LIN {X 0,Y 175.493,Z 504.64,A -85,B 0,C 180,E1 -23519.914,E2 -23519.914} C_VEL
LIN {X 0,Y 175.421,Z 500.697,A -85,B 0,C 180,E1 -23521.362,E2 -23521.362} C_VEL
LIN {X 0,Y 174.535,Z 496.874,A -85,B 0,C 180,E1 -23522.837,E2 -23522.837} C_VEL
LIN {X 0,Y 173.048,Z 491.549,A -85,B 0,C 180,E1 -23524.809,E2 -23524.809} C_VEL
LIN {X 0,Y 172.478,Z 487.181,A -85,B 0,C 180,E1 -23526.194,E2 -23526.194} C_VEL
LIN {X 0,Y 172.504,Z 485.618,A -85,B 0,C 180,E1 -23526.619,E2 -23526.619} C_VEL
LIN {X 0,Y 172.737,Z 474.589,A -85,B 0,C 180,E1 -23529.373,E2 -23529.373} C_VEL
LIN {X 0,Y 172.189,Z 465.013,A -85,B 0,C 180,E1 -23531.567,E2 -23531.567} C_VEL
LIN {X 0,Y 171.174,Z 457.609,A -85,B 0,C 180,E1 -23533.216,E2 -23533.216} C_VEL
LIN {X 0,Y 168.739,Z 450.808,A -85,B 0,C 180,E1 -23535.077,E2 -23535.077} C_VEL
LIN {X 0,Y 164.618,Z 441.913,A -85,B 0,C 180,E1 -23537.724,E2 -23537.724} C_VEL
LIN {X 0,Y 162.473,Z 437.771,A -85,B 0,C 180,E1 -23539.043,E2 -23539.043} C_VEL
LIN {X 0,Y 161.542,Z 436.333,A -85,B 0,C 180,E1 -23539.565,E2 -23539.565} C_VEL
LIN {X 0,Y 159.595,Z 433.029,A -85,B 0,C 180,E1 -23540.726,E2 -23540.726} C_VEL
LIN {X 0,Y 159.065,Z 431.216,A -85,B 0,C 180,E1 -23541.182,E2 -23541.182} C_VEL
LIN {X 0,Y 158.472,Z 427.771,A -85,B 0,C 180,E1 -23547.418,E2 -23547.418} C_VEL
LIN {X 0,Y 158.056,Z 424.721,A -85,B 0,C 180,E1 -23553.599,E2 -23553.599} C_VEL
LIN {X 0,Y 157.656,Z 422.287,A -85,B 0,C 180,E1 -23559.413,E2 -23559.413} C_VEL
LIN {X 0,Y 157.505,Z 421.4,A -85,B 0,C 180,E1 -23561.799,E2 -23561.799} C_VEL
LIN {X 0,Y 157.48,Z 420.87,A -85,B 0,C 180,E1 -23564.469,E2 -23564.469} C_VEL
LIN {X 0,Y 157.774,Z 420.833,A -85,B 0,C 180,E1 -23569.736,E2 -23569.736} C_VEL
LIN {X 0,Y 157.827,Z 420.827,A -85,B 0,C 180,E1 -23572.323,E2 -23572.323} C_VEL
LIN {X 0,Y 158.262,Z 420.771,A -85,B 0,C 180,E1 -23580,E2 -23580} C_VEL
LIN {X 0,Y 157.827,Z 420.823,A -85,B 0,C 180,E1 -23587.677,E2 -23587.677} C_VEL
LIN {X 0,Y 157.707,Z 420.841,A -85,B 0,C 180,E1 -23591.363,E2 -23591.363} C_VEL
LIN {X 0,Y 157.48,Z 420.866,A -85,B 0,C 180,E1 -23595.532,E2 -23595.532} C_VEL
LIN {X 0,Y 157.369,Z 420.882,A -85,B 0,C 180,E1 -23600.933,E2 -23600.933} C_VEL
LIN {X 0,Y 157.31,Z 420.887,A -85,B 0,C 180,E1 -23606.681,E2 -23606.681} C_VEL
LIN {X 0,Y 157.277,Z 420.885,A -85,B 0,C 180,E1 -23612.427,E2 -23612.427} C_VEL
LIN {X 0,Y 157.252,Z 420.892,A -85,B 0,C 180,E1 -23617.475,E2 -23617.475} C_VEL
LIN {X 0,Y 157.23,Z 421.026,A -85,B 0,C 180,E1 -23618.265,E2 -23618.265} C_VEL
LIN {X 0,Y 158.236,Z 423.75,A -85,B 0,C 180,E1 -23619.044,E2 -23619.044} C_VEL
LIN {X 0,Y 160.601,Z 426.337,A -85,B 0,C 180,E1 -23620.395,E2 -23620.395} C_VEL
LIN {X 0,Y 162.443,Z 429.537,A -85,B 0,C 180,E1 -23621.594,E2 -23621.594} C_VEL
LIN {X 0,Y 163.808,Z 431.474,A -85,B 0,C 180,E1 -23622.408,E2 -23622.408} C_VEL
LIN {X 0,Y 168.225,Z 439.084,A -85,B 0,C 180,E1 -23625.253,E2 -23625.253} C_VEL
LIN {X 0,Y 171.385,Z 446.088,A -85,B 0,C 180,E1 -23627.572,E2 -23627.572} C_VEL
LIN {X 0,Y 174.009,Z 454.383,A -85,B 0,C 180,E1 -23630.12,E2 -23630.12} C_VEL
LIN {X 0,Y 175.758,Z 463.088,A -85,B 0,C 180,E1 -23632.727,E2 -23632.727} C_VEL
LIN {X 0,Y 176.597,Z 472.445,A -85,B 0,C 180,E1 -23635.6,E2 -23635.6} C_VEL
LIN {X 0,Y 176.668,Z 474.207,A -85,B 0,C 180,E1 -23636.156,E2 -23636.156} C_VEL
LIN {X 0,Y 174.39,Z 481.217,A -85,B 0,C 180,E1 -23638.023,E2 -23638.023} C_VEL
LIN {X 0,Y 170.562,Z 490.741,A -85,B 0,C 180,E1 -23641.043,E2 -23641.043} C_VEL
LIN {X 0,Y 166.711,Z 498.951,A -85,B 0,C 180,E1 -23644.399,E2 -23644.399} C_VEL
LIN {X 0,Y 164.054,Z 504.551,A -85,B 0,C 180,E1 -23647.322,E2 -23647.322} C_VEL
LIN {X 0,Y 161.243,Z 510.012,A -85,B 0,C 180,E1 -23650.92,E2 -23650.92} C_VEL
LIN {X 0,Y 158.999,Z 514.292,A -85,B 0,C 180,E1 -23654.621,E2 -23654.621} C_VEL
LIN {X 0,Y 157.864,Z 516.551,A -85,B 0,C 180,E1 -23657.139,E2 -23657.139} C_VEL
LIN {X 0,Y 156.746,Z 518.873,A -85,B 0,C 180,E1 -23660.546,E2 -23660.546} C_VEL
LIN {X 0,Y 155.819,Z 520.739,A -85,B 0,C 180,E1 -23664.825,E2 -23664.825} C_VEL
LIN {X 0,Y 155.405,Z 521.567,A -85,B 0,C 180,E1 -23670,E2 -23670} C_VEL
LIN {X 0,Y 155.514,Z 521.37,A -85,B 0,C 180,E1 -23672.59,E2 -23672.59} C_VEL
LIN {X 0,Y 155.811,Z 520.787,A -85,B 0,C 180,E1 -23675.176,E2 -23675.176} C_VEL
LIN {X 0,Y 156.94,Z 518.483,A -85,B 0,C 180,E1 -23680.319,E2 -23680.319} C_VEL
LIN {X 0,Y 158.342,Z 515.638,A -85,B 0,C 180,E1 -23684.13,E2 -23684.13} C_VEL
LIN {X 0,Y 160.383,Z 511.769,A -85,B 0,C 180,E1 -23687.863,E2 -23687.863} C_VEL
LIN {X 0,Y 162.981,Z 506.773,A -85,B 0,C 180,E1 -23691.502,E2 -23691.502} C_VEL
LIN {X 0,Y 166.065,Z 500.477,A -85,B 0,C 180,E1 -23695.038,E2 -23695.038} C_VEL
LIN {X 0,Y 169.842,Z 492.583,A -85,B 0,C 180,E1 -23698.416,E2 -23698.416} C_VEL
LIN {X 0,Y 173.954,Z 482.769,A -85,B 0,C 180,E1 -23701.684,E2 -23701.684} C_VEL
LIN {X 0,Y 176.747,Z 474.731,A -85,B 0,C 180,E1 -23703.827,E2 -23703.827} C_VEL
LIN {X 0,Y 176.346,Z 467.155,A -85,B 0,C 180,E1 -23706.194,E2 -23706.194} C_VEL
LIN {X 0,Y 174.874,Z 457.677,A -85,B 0,C 180,E1 -23709.05,E2 -23709.05} C_VEL
LIN {X 0,Y 172.59,Z 449.442,A -85,B 0,C 180,E1 -23711.56,E2 -23711.56} C_VEL
LIN {X 0,Y 170.161,Z 443.217,A -85,B 0,C 180,E1 -23713.554,E2 -23713.554} C_VEL
LIN {X 0,Y 165.724,Z 434.544,A -85,B 0,C 180,E1 -23716.601,E2 -23716.601} C_VEL
LIN {X 0,Y 163.507,Z 430.878,A -85,B 0,C 180,E1 -23718.016,E2 -23718.016} C_VEL
LIN {X 0,Y 160.947,Z 427.183,A -85,B 0,C 180,E1 -23719.565,E2 -23719.565} C_VEL
LIN {X 0,Y 160.394,Z 425.942,A -85,B 0,C 180,E1 -23719.971,E2 -23719.971} C_VEL
LIN {X 0,Y 158.165,Z 423.621,A -85,B 0,C 180,E1 -23721.234,E2 -23721.234} C_VEL
LIN {X 0,Y 157.222,Z 420.897,A -85,B 0,C 180,E1 -23722.046,E2 -23722.046} C_VEL
LIN {X 0,Y 157.292,Z 420.884,A -85,B 0,C 180,E1 -23724.489,E2 -23724.489} C_VEL
LIN {X 0,Y 157.296,Z 420.89,A -85,B 0,C 180,E1 -23728.096,E2 -23728.096} C_VEL
LIN {X 0,Y 157.317,Z 420.889,A -85,B 0,C 180,E1 -23733.465,E2 -23733.465} C_VEL
LIN {X 0,Y 157.395,Z 420.879,A -85,B 0,C 180,E1 -23739.669,E2 -23739.669} C_VEL
LIN {X 0,Y 157.476,Z 420.869,A -85,B 0,C 180,E1 -23744.468,E2 -23744.468} C_VEL
LIN {X 0,Y 157.692,Z 420.84,A -85,B 0,C 180,E1 -23749.731,E2 -23749.731} C_VEL
LIN {X 0,Y 157.77,Z 420.831,A -85,B 0,C 180,E1 -23752.32,E2 -23752.32} C_VEL
LIN {X 0,Y 158.261,Z 420.776,A -85,B 0,C 180,E1 -23760,E2 -23760} C_VEL
LIN {X 0,Y 157.828,Z 420.829,A -85,B 0,C 180,E1 -23767.677,E2 -23767.677} C_VEL
LIN {X 0,Y 157.72,Z 420.838,A -85,B 0,C 180,E1 -23771.383,E2 -23771.383} C_VEL
LIN {X 0,Y 157.489,Z 420.866,A -85,B 0,C 180,E1 -23775.531,E2 -23775.531} C_VEL
LIN {X 0,Y 157.542,Z 421.446,A -85,B 0,C 180,E1 -23778.196,E2 -23778.196} C_VEL
LIN {X 0,Y 157.82,Z 423.583,A -85,B 0,C 180,E1 -23783.627,E2 -23783.627} C_VEL
LIN {X 0,Y 158.101,Z 425.177,A -85,B 0,C 180,E1 -23787.244,E2 -23787.244} C_VEL
LIN {X 0,Y 158.474,Z 427.834,A -85,B 0,C 180,E1 -23792.582,E2 -23792.582} C_VEL
LIN {X 0,Y 159.063,Z 431.245,A -85,B 0,C 180,E1 -23798.717,E2 -23798.717} C_VEL
LIN {X 0,Y 160.489,Z 434.863,A -85,B 0,C 180,E1 -23799.723,E2 -23799.723} C_VEL
LIN {X 0,Y 162.468,Z 437.655,A -85,B 0,C 180,E1 -23800.825,E2 -23800.825} C_VEL
LIN {X 0,Y 164.462,Z 441.653,A -85,B 0,C 180,E1 -23802.073,E2 -23802.073} C_VEL
LIN {X 0,Y 165.475,Z 443.522,A -85,B 0,C 180,E1 -23802.676,E2 -23802.676} C_VEL
LIN {X 0,Y 168.043,Z 449.265,A -85,B 0,C 180,E1 -23804.365,E2 -23804.365} C_VEL
LIN {X 0,Y 170.827,Z 456.275,A -85,B 0,C 180,E1 -23806.35,E2 -23806.35} C_VEL
LIN {X 0,Y 172.062,Z 463.231,A -85,B 0,C 180,E1 -23807.965,E2 -23807.965} C_VEL
LIN {X 0,Y 172.805,Z 473.587,A -85,B 0,C 180,E1 -23810.33,E2 -23810.33} C_VEL
LIN {X 0,Y 172.705,Z 483.558,A -85,B 0,C 180,E1 -23812.784,E2 -23812.784} C_VEL
LIN {X 0,Y 171.722,Z 494.309,A -85,B 0,C 180,E1 -23815.754,E2 -23815.754} C_VEL
LIN {X 0,Y 170.269,Z 502.262,A -85,B 0,C 180,E1 -23818.246,E2 -23818.246} C_VEL
LIN {X 0,Y 168.438,Z 507.397,A -85,B 0,C 180,E1 -23819.953,E2 -23819.953} C_VEL
LIN {X 0,Y 165.157,Z 514.724,A -85,B 0,C 180,E1 -23822.777,E2 -23822.777} C_VEL
LIN {X 0,Y 162.483,Z 520.901,A -85,B 0,C 180,E1 -23825.773,E2 -23825.773} C_VEL
LIN {X 0,Y 159.679,Z 526.854,A -85,B 0,C 180,E1 -23829.383,E2 -23829.383} C_VEL
LIN {X 0,Y 157.532,Z 531.619,A -85,B 0,C 180,E1 -23833.142,E2 -23833.142} C_VEL
LIN {X 0,Y 156.082,Z 535.276,A -85,B 0,C 180,E1 -23836.989,E2 -23836.989} C_VEL
LIN {X 0,Y 155.465,Z 537.169,A -85,B 0,C 180,E1 -23839.582,E2 -23839.582} C_VEL
LIN {X 0,Y 155.141,Z 538.598,A -85,B 0,C 180,E1 -23842.189,E2 -23842.189} C_VEL
LIN {X 0,Y 155.009,Z 539.965,A -85,B 0,C 180,E1 -23845.92,E2 -23845.92} C_VEL
LIN {X 0,Y 155.237,Z 540.486,A -85,B 0,C 180,E1 -23850,E2 -23850} C_VEL
LIN {X 0,Y 155.013,Z 539.948,A -85,B 0,C 180,E1 -23854.1,E2 -23854.1} C_VEL
LIN {X 0,Y 155.113,Z 538.571,A -85,B 0,C 180,E1 -23857.812,E2 -23857.812} C_VEL
LIN {X 0,Y 155.463,Z 537.132,A -85,B 0,C 180,E1 -23860.418,E2 -23860.418} C_VEL
LIN {X 0,Y 156.466,Z 534.131,A -85,B 0,C 180,E1 -23864.302,E2 -23864.302} C_VEL
LIN {X 0,Y 158.189,Z 530.096,A -85,B 0,C 180,E1 -23868.119,E2 -23868.119} C_VEL
LIN {X 0,Y 161.039,Z 523.913,A -85,B 0,C 180,E1 -23872.449,E2 -23872.449} C_VEL
LIN {X 0,Y 164.023,Z 517.168,A -85,B 0,C 180,E1 -23876.052,E2 -23876.052} C_VEL
LIN {X 0,Y 167.699,Z 508.823,A -85,B 0,C 180,E1 -23879.5,E2 -23879.5} C_VEL
LIN {X 0,Y 169.803,Z 503.886,A -85,B 0,C 180,E1 -23881.156,E2 -23881.156} C_VEL
LIN {X 0,Y 171.491,Z 495.166,A -85,B 0,C 180,E1 -23883.944,E2 -23883.944} C_VEL
LIN {X 0,Y 172.504,Z 485.618,A -85,B 0,C 180,E1 -23886.619,E2 -23886.619} C_VEL
LIN {X 0,Y 172.159,Z 481.183,A -85,B 0,C 180,E1 -23887.899,E2 -23887.899} C_VEL
LIN {X 0,Y 170.903,Z 477.034,A -85,B 0,C 180,E1 -23889.266,E2 -23889.266} C_VEL
LIN {X 0,Y 167.544,Z 468.986,A -85,B 0,C 180,E1 -23892.064,E2 -23892.064} C_VEL
LIN {X 0,Y 166.046,Z 462.962,A -85,B 0,C 180,E1 -23893.79,E2 -23893.79} C_VEL
LIN {X 0,Y 165.199,Z 458.874,A -85,B 0,C 180,E1 -23894.864,E2 -23894.864} C_VEL
LIN {X 0,Y 162.424,Z 451.6,A -85,B 0,C 180,E1 -23897.123,E2 -23897.123} C_VEL
LIN {X 0,Y 159.982,Z 446.385,A -85,B 0,C 180,E1 -23898.885,E2 -23898.885} C_VEL
LIN {X 0,Y 157.628,Z 441.579,A -85,B 0,C 180,E1 -23900.554,E2 -23900.554} C_VEL
LIN {X 0,Y 155.555,Z 437.698,A -85,B 0,C 180,E1 -23902.001,E2 -23902.001} C_VEL
LIN {X 0,Y 154.89,Z 436.44,A -85,B 0,C 180,E1 -23902.456,E2 -23902.456} C_VEL
LIN {X 0,Y 152.505,Z 433.06,A -85,B 0,C 180,E1 -23904.015,E2 -23904.015} C_VEL
LIN {X 0,Y 151.729,Z 430.582,A -85,B 0,C 180,E1 -23904.722,E2 -23904.722} C_VEL
LIN {X 0,Y 151.32,Z 428.28,A -85,B 0,C 180,E1 -23909.277,E2 -23909.277} C_VEL
LIN {X 0,Y 151.168,Z 426.831,A -85,B 0,C 180,E1 -23912.295,E2 -23912.295} C_VEL
LIN {X 0,Y 150.769,Z 424.399,A -85,B 0,C 180,E1 -23918.105,E2 -23918.105} C_VEL
LIN {X 0,Y 150.494,Z 422.416,A -85,B 0,C 180,E1 -23923.728,E2 -23923.728} C_VEL
LIN {X 0,Y 150.466,Z 421.744,A -85,B 0,C 180,E1 -23926.494,E2 -23926.494} C_VEL
LIN {X 0,Y 150.697,Z 421.715,A -85,B 0,C 180,E1 -23929.249,E2 -23929.249} C_VEL
LIN {X 0,Y 150.765,Z 421.706,A -85,B 0,C 180,E1 -23931.961,E2 -23931.961} C_VEL
LIN {X 0,Y 151.222,Z 421.648,A -85,B 0,C 180,E1 -23940,E2 -23940} C_VEL
LIN {X 0,Y 150.765,Z 421.704,A -85,B 0,C 180,E1 -23948.039,E2 -23948.039} C_VEL
LIN {X 0,Y 150.637,Z 421.722,A -85,B 0,C 180,E1 -23951.546,E2 -23951.546} C_VEL
LIN {X 0,Y 150.385,Z 421.75,A -85,B 0,C 180,E1 -23956.284,E2 -23956.284} C_VEL
LIN {X 0,Y 150.351,Z 421.756,A -85,B 0,C 180,E1 -23960.791,E2 -23960.791} C_VEL
LIN {X 0,Y 150.242,Z 421.768,A -85,B 0,C 180,E1 -23967.28,E2 -23967.28} C_VEL
LIN {X 0,Y 150.217,Z 421.764,A -85,B 0,C 180,E1 -23972.633,E2 -23972.633} C_VEL
LIN {X 0,Y 150.234,Z 421.892,A -85,B 0,C 180,E1 -23974.76,E2 -23974.76} C_VEL
LIN {X 0,Y 151.187,Z 424.529,A -85,B 0,C 180,E1 -23975.628,E2 -23975.628} C_VEL
LIN {X 0,Y 153.348,Z 426.792,A -85,B 0,C 180,E1 -23977.056,E2 -23977.056} C_VEL
LIN {X 0,Y 155.822,Z 430.828,A -85,B 0,C 180,E1 -23978.864,E2 -23978.864} C_VEL
LIN {X 0,Y 156.885,Z 432.163,A -85,B 0,C 180,E1 -23979.566,E2 -23979.566} C_VEL
LIN {X 0,Y 160.888,Z 438.893,A -85,B 0,C 180,E1 -23982.446,E2 -23982.446} C_VEL
LIN {X 0,Y 164.275,Z 445.344,A -85,B 0,C 180,E1 -23984.992,E2 -23984.992} C_VEL
LIN {X 0,Y 166.93,Z 452.435,A -85,B 0,C 180,E1 -23987.46,E2 -23987.46} C_VEL
LIN {X 0,Y 168.941,Z 460.421,A -85,B 0,C 180,E1 -23990.069,E2 -23990.069} C_VEL
LIN {X 0,Y 170.032,Z 468.449,A -85,B 0,C 180,E1 -23992.662,E2 -23992.662} C_VEL
LIN {X 0,Y 170.291,Z 476.562,A -85,B 0,C 180,E1 -23995.361,E2 -23995.361} C_VEL
LIN {X 0,Y 166.541,Z 486.299,A -85,B 0,C 180,E1 -23998.163,E2 -23998.163} C_VEL
LIN {X 0,Y 162.992,Z 494.122,A -85,B 0,C 180,E1 -24000.982,E2 -24000.982} C_VEL
LIN {X 0,Y 159.238,Z 501.757,A -85,B 0,C 180,E1 -24004.512,E2 -24004.512} C_VEL
LIN {X 0,Y 155.5,Z 508.765,A -85,B 0,C 180,E1 -24008.804,E2 -24008.804} C_VEL
LIN {X 0,Y 152.899,Z 513.427,A -85,B 0,C 180,E1 -24012.616,E2 -24012.616} C_VEL
LIN {X 0,Y 150.96,Z 516.984,A -85,B 0,C 180,E1 -24016.54,E2 -24016.54} C_VEL
LIN {X 0,Y 149.624,Z 519.54,A -85,B 0,C 180,E1 -24020.539,E2 -24020.539} C_VEL
LIN {X 0,Y 148.769,Z 521.17,A -85,B 0,C 180,E1 -24024.579,E2 -24024.579} C_VEL
LIN {X 0,Y 148.465,Z 521.771,A -85,B 0,C 180,E1 -24027.287,E2 -24027.287} C_VEL
LIN {X 0,Y 148.346,Z 521.997,A -85,B 0,C 180,E1 -24030,E2 -24030} C_VEL
LIN {X 0,Y 148.462,Z 521.8,A -85,B 0,C 180,E1 -24032.714,E2 -24032.714} C_VEL
LIN {X 0,Y 148.76,Z 521.218,A -85,B 0,C 180,E1 -24035.422,E2 -24035.422} C_VEL
LIN {X 0,Y 149.979,Z 518.913,A -85,B 0,C 180,E1 -24040.804,E2 -24040.804} C_VEL
LIN {X 0,Y 151.475,Z 516.069,A -85,B 0,C 180,E1 -24044.785,E2 -24044.785} C_VEL
LIN {X 0,Y 153.644,Z 512.2,A -85,B 0,C 180,E1 -24048.675,E2 -24048.675} C_VEL
LIN {X 0,Y 156.409,Z 507.203,A -85,B 0,C 180,E1 -24052.454,E2 -24052.454} C_VEL
LIN {X 0,Y 159.667,Z 500.906,A -85,B 0,C 180,E1 -24056.115,E2 -24056.115} C_VEL
LIN {X 0,Y 163.653,Z 493.011,A -85,B 0,C 180,E1 -24059.595,E2 -24059.595} C_VEL
LIN {X 0,Y 167.954,Z 483.198,A -85,B 0,C 180,E1 -24062.956,E2 -24062.956} C_VEL
LIN {X 0,Y 170.483,Z 476.31,A -85,B 0,C 180,E1 -24064.859,E2 -24064.859} C_VEL
LIN {X 0,Y 170.175,Z 468.722,A -85,B 0,C 180,E1 -24067.401,E2 -24067.401} C_VEL
LIN {X 0,Y 168.987,Z 460.08,A -85,B 0,C 180,E1 -24070.194,E2 -24070.194} C_VEL
LIN {X 0,Y 167.089,Z 452.794,A -85,B 0,C 180,E1 -24072.6,E2 -24072.6} C_VEL
LIN {X 0,Y 164.806,Z 446.556,A -85,B 0,C 180,E1 -24074.781,E2 -24074.781} C_VEL
LIN {X 0,Y 161.086,Z 439.296,A -85,B 0,C 180,E1 -24077.618,E2 -24077.618} C_VEL
LIN {X 0,Y 156.396,Z 431.427,A -85,B 0,C 180,E1 -24081.014,E2 -24081.014} C_VEL
LIN {X 0,Y 154.307,Z 428.597,A -85,B 0,C 180,E1 -24082.434,E2 -24082.434} C_VEL
LIN {X 0,Y 153.487,Z 426.898,A -85,B 0,C 180,E1 -24083.103,E2 -24083.103} C_VEL
LIN {X 0,Y 151.343,Z 424.737,A -85,B 0,C 180,E1 -24084.516,E2 -24084.516} C_VEL
LIN {X 0,Y 150.258,Z 422.177,A -85,B 0,C 180,E1 -24085.45,E2 -24085.45} C_VEL
LIN {X 0,Y 150.206,Z 421.769,A -85,B 0,C 180,E1 -24085.64,E2 -24085.64} C_VEL
LIN {X 0,Y 150.209,Z 421.775,A -85,B 0,C 180,E1 -24089.024,E2 -24089.024} C_VEL
LIN {X 0,Y 150.243,Z 421.768,A -85,B 0,C 180,E1 -24092.721,E2 -24092.721} C_VEL
LIN {X 0,Y 150.352,Z 421.757,A -85,B 0,C 180,E1 -24099.209,E2 -24099.209} C_VEL
LIN {X 0,Y 150.382,Z 421.75,A -85,B 0,C 180,E1 -24103.715,E2 -24103.715} C_VEL
LIN {X 0,Y 150.615,Z 421.721,A -85,B 0,C 180,E1 -24109.243,E2 -24109.243} C_VEL
LIN {X 0,Y 150.707,Z 421.711,A -85,B 0,C 180,E1 -24111.958,E2 -24111.958} C_VEL
LIN {X 0,Y 151.221,Z 421.654,A -85,B 0,C 180,E1 -24120,E2 -24120} C_VEL
LIN {X 0,Y 150.767,Z 421.709,A -85,B 0,C 180,E1 -24128.039,E2 -24128.039} C_VEL
LIN {X 0,Y 150.645,Z 421.719,A -85,B 0,C 180,E1 -24131.56,E2 -24131.56} C_VEL
LIN {X 0,Y 150.47,Z 421.741,A -85,B 0,C 180,E1 -24133.505,E2 -24133.505} C_VEL
LIN {X 0,Y 150.665,Z 423.414,A -85,B 0,C 180,E1 -24139.058,E2 -24139.058} C_VEL
LIN {X 0,Y 150.946,Z 425.635,A -85,B 0,C 180,E1 -24144.774,E2 -24144.774} C_VEL
LIN {X 0,Y 151.185,Z 427.018,A -85,B 0,C 180,E1 -24147.963,E2 -24147.963} C_VEL
LIN {X 0,Y 151.646,Z 430.268,A -85,B 0,C 180,E1 -24154.592,E2 -24154.592} C_VEL
LIN {X 0,Y 151.724,Z 430.738,A -85,B 0,C 180,E1 -24155.178,E2 -24155.178} C_VEL
LIN {X 0,Y 152.952,Z 433.942,A -85,B 0,C 180,E1 -24156.168,E2 -24156.168} C_VEL
LIN {X 0,Y 155.39,Z 437.231,A -85,B 0,C 180,E1 -24157.73,E2 -24157.73} C_VEL
LIN {X 0,Y 157.426,Z 441.33,A -85,B 0,C 180,E1 -24159.196,E2 -24159.196} C_VEL
LIN {X 0,Y 158.706,Z 443.64,A -85,B 0,C 180,E1 -24160.053,E2 -24160.053} C_VEL
LIN {X 0,Y 161.186,Z 448.748,A -85,B 0,C 180,E1 -24161.826,E2 -24161.826} C_VEL
LIN {X 0,Y 164.43,Z 456.664,A -85,B 0,C 180,E1 -24164.36,E2 -24164.36} C_VEL
LIN {X 0,Y 165.782,Z 460.967,A -85,B 0,C 180,E1 -24165.615,E2 -24165.615} C_VEL
LIN {X 0,Y 166.735,Z 470.398,A -85,B 0,C 180,E1 -24167.933,E2 -24167.933} C_VEL
LIN {X 0,Y 166.739,Z 481.622,A -85,B 0,C 180,E1 -24170.783,E2 -24170.783} C_VEL
LIN {X 0,Y 165.823,Z 491.754,A -85,B 0,C 180,E1 -24173.636,E2 -24173.636} C_VEL
LIN {X 0,Y 164.504,Z 499.99,A -85,B 0,C 180,E1 -24176.262,E2 -24176.262} C_VEL
LIN {X 0,Y 163.014,Z 505.323,A -85,B 0,C 180,E1 -24178.12,E2 -24178.12} C_VEL
LIN {X 0,Y 158.822,Z 514.29,A -85,B 0,C 180,E1 -24181.595,E2 -24181.595} C_VEL
LIN {X 0,Y 155.634,Z 521.247,A -85,B 0,C 180,E1 -24185.126,E2 -24185.126} C_VEL
LIN {X 0,Y 153.002,Z 526.42,A -85,B 0,C 180,E1 -24188.44,E2 -24188.44} C_VEL
LIN {X 0,Y 150.706,Z 531.185,A -85,B 0,C 180,E1 -24192.355,E2 -24192.355} C_VEL
LIN {X 0,Y 149.123,Z 534.841,A -85,B 0,C 180,E1 -24196.37,E2 -24196.37} C_VEL
LIN {X 0,Y 148.469,Z 536.736,A -85,B 0,C 180,E1 -24199.085,E2 -24199.085} C_VEL
LIN {X 0,Y 148.07,Z 538.164,A -85,B 0,C 180,E1 -24201.813,E2 -24201.813} C_VEL
LIN {X 0,Y 147.94,Z 539.595,A -85,B 0,C 180,E1 -24206.05,E2 -24206.05} C_VEL
LIN {X 0,Y 148.153,Z 540.054,A -85,B 0,C 180,E1 -24210,E2 -24210} C_VEL
LIN {X 0,Y 147.934,Z 539.59,A -85,B 0,C 180,E1 -24213.916,E2 -24213.916} C_VEL
LIN {X 0,Y 148.046,Z 538.136,A -85,B 0,C 180,E1 -24218.187,E2 -24218.187} C_VEL
LIN {X 0,Y 148.468,Z 536.698,A -85,B 0,C 180,E1 -24220.915,E2 -24220.915} C_VEL
LIN {X 0,Y 149.564,Z 533.695,A -85,B 0,C 180,E1 -24224.978,E2 -24224.978} C_VEL
LIN {X 0,Y 151.409,Z 529.659,A -85,B 0,C 180,E1 -24228.961,E2 -24228.961} C_VEL
LIN {X 0,Y 154.493,Z 523.478,A -85,B 0,C 180,E1 -24233.456,E2 -24233.456} C_VEL
LIN {X 0,Y 157.656,Z 516.732,A -85,B 0,C 180,E1 -24237.189,E2 -24237.189} C_VEL
LIN {X 0,Y 161.544,Z 508.387,A -85,B 0,C 180,E1 -24240.743,E2 -24240.743} C_VEL
LIN {X 0,Y 163.59,Z 503.438,A -85,B 0,C 180,E1 -24242.48,E2 -24242.48} C_VEL
LIN {X 0,Y 165.321,Z 494.743,A -85,B 0,C 180,E1 -24245.383,E2 -24245.383} C_VEL
LIN {X 0,Y 166.4,Z 485.318,A -85,B 0,C 180,E1 -24248.148,E2 -24248.148} C_VEL
LIN {X 0,Y 166.763,Z 474.342,A -85,B 0,C 180,E1 -24251.02,E2 -24251.02} C_VEL
LIN {X 0,Y 166.149,Z 463.815,A -85,B 0,C 180,E1 -24253.583,E2 -24253.583} C_VEL
LIN {X 0,Y 166.046,Z 462.962,A -85,B 0,C 180,E1 -24253.79,E2 -24253.79} C_VEL
LIN {X 0,Y 165.299,Z 460.01,A -85,B 0,C 180,E1 -24254.631,E2 -24254.631} C_VEL
LIN {X 0,Y 163.174,Z 456.37,A -85,B 0,C 180,E1 -24256.067,E2 -24256.067} C_VEL
LIN {X 0,Y 160.391,Z 453.439,A -85,B 0,C 180,E1 -24257.617,E2 -24257.617} C_VEL
LIN {X 0,Y 154.426,Z 447.845,A -85,B 0,C 180,E1 -24260.975,E2 -24260.975} C_VEL
LIN {X 0,Y 152.812,Z 445.559,A -85,B 0,C 180,E1 -24262.089,E2 -24262.089} C_VEL
LIN {X 0,Y 150.995,Z 441.721,A -85,B 0,C 180,E1 -24263.598,E2 -24263.598} C_VEL
LIN {X 0,Y 148.744,Z 437.9,A -85,B 0,C 180,E1 -24265.357,E2 -24265.357} C_VEL
LIN {X 0,Y 147.886,Z 436.021,A -85,B 0,C 180,E1 -24266.099,E2 -24266.099} C_VEL
LIN {X 0,Y 145.416,Z 432.796,A -85,B 0,C 180,E1 -24267.986,E2 -24267.986} C_VEL
LIN {X 0,Y 144.374,Z 429.792,A -85,B 0,C 180,E1 -24269.058,E2 -24269.058} C_VEL
LIN {X 0,Y 144.059,Z 427.599,A -85,B 0,C 180,E1 -24273.956,E2 -24273.956} C_VEL
LIN {X 0,Y 143.761,Z 425.302,A -85,B 0,C 180,E1 -24279.989,E2 -24279.989} C_VEL
LIN {X 0,Y 143.529,Z 423.451,A -85,B 0,C 180,E1 -24285.828,E2 -24285.828} C_VEL
LIN {X 0,Y 143.624,Z 422.621,A -85,B 0,C 180,E1 -24288.713,E2 -24288.713} C_VEL
LIN {X 0,Y 143.688,Z 422.587,A -85,B 0,C 180,E1 -24291.562,E2 -24291.562} C_VEL
LIN {X 0,Y 144.181,Z 422.525,A -85,B 0,C 180,E1 -24300,E2 -24300} C_VEL
LIN {X 0,Y 143.687,Z 422.588,A -85,B 0,C 180,E1 -24308.438,E2 -24308.438} C_VEL
LIN {X 0,Y 143.573,Z 422.602,A -85,B 0,C 180,E1 -24311.758,E2 -24311.758} C_VEL
LIN {X 0,Y 143.318,Z 422.633,A -85,B 0,C 180,E1 -24317.111,E2 -24317.111} C_VEL
LIN {X 0,Y 143.277,Z 422.636,A -85,B 0,C 180,E1 -24321.253,E2 -24321.253} C_VEL
LIN {X 0,Y 143.189,Z 422.649,A -85,B 0,C 180,E1 -24327.936,E2 -24327.936} C_VEL
LIN {X 0,Y 143.139,Z 422.68,A -85,B 0,C 180,E1 -24330.42,E2 -24330.42} C_VEL
LIN {X 0,Y 144.036,Z 425.274,A -85,B 0,C 180,E1 -24331.432,E2 -24331.432} C_VEL
LIN {X 0,Y 146.042,Z 427.52,A -85,B 0,C 180,E1 -24333.062,E2 -24333.062} C_VEL
LIN {X 0,Y 147.03,Z 428.412,A -85,B 0,C 180,E1 -24333.822,E2 -24333.822} C_VEL
LIN {X 0,Y 148.875,Z 431.662,A -85,B 0,C 180,E1 -24335.434,E2 -24335.434} C_VEL
LIN {X 0,Y 150.282,Z 433.284,A -85,B 0,C 180,E1 -24336.499,E2 -24336.499} C_VEL
LIN {X 0,Y 151.961,Z 436.253,A -85,B 0,C 180,E1 -24337.919,E2 -24337.919} C_VEL
LIN {X 0,Y 154.914,Z 440.993,A -85,B 0,C 180,E1 -24340.277,E2 -24340.277} C_VEL
LIN {X 0,Y 158.568,Z 448.092,A -85,B 0,C 180,E1 -24343.393,E2 -24343.393} C_VEL
LIN {X 0,Y 160.834,Z 453.765,A -85,B 0,C 180,E1 -24345.641,E2 -24345.641} C_VEL
LIN {X 0,Y 162.963,Z 462.342,A -85,B 0,C 180,E1 -24348.697,E2 -24348.697} C_VEL
LIN {X 0,Y 163.963,Z 470.103,A -85,B 0,C 180,E1 -24351.399,E2 -24351.399} C_VEL
LIN {X 0,Y 164.171,Z 477.153,A -85,B 0,C 180,E1 -24353.919,E2 -24353.919} C_VEL
LIN {X 0,Y 163.706,Z 479.185,A -85,B 0,C 180,E1 -24354.538,E2 -24354.538} C_VEL
LIN {X 0,Y 159.832,Z 488.41,A -85,B 0,C 180,E1 -24357.409,E2 -24357.409} C_VEL
LIN {X 0,Y 155.395,Z 497.277,A -85,B 0,C 180,E1 -24360.91,E2 -24360.91} C_VEL
LIN {X 0,Y 151.696,Z 504.396,A -85,B 0,C 180,E1 -24364.625,E2 -24364.625} C_VEL
LIN {X 0,Y 148.928,Z 509.198,A -85,B 0,C 180,E1 -24367.82,E2 -24367.82} C_VEL
LIN {X 0,Y 146.163,Z 513.859,A -85,B 0,C 180,E1 -24371.788,E2 -24371.788} C_VEL
LIN {X 0,Y 144.089,Z 517.416,A -85,B 0,C 180,E1 -24375.885,E2 -24375.885} C_VEL
LIN {X 0,Y 142.562,Z 520.132,A -85,B 0,C 180,E1 -24380.388,E2 -24380.388} C_VEL
LIN {X 0,Y 141.723,Z 521.602,A -85,B 0,C 180,E1 -24384.308,E2 -24384.308} C_VEL
LIN {X 0,Y 141.288,Z 522.427,A -85,B 0,C 180,E1 -24390,E2 -24390} C_VEL
LIN {X 0,Y 141.389,Z 522.231,A -85,B 0,C 180,E1 -24392.849,E2 -24392.849} C_VEL
LIN {X 0,Y 141.713,Z 521.649,A -85,B 0,C 180,E1 -24395.693,E2 -24395.693} C_VEL
LIN {X 0,Y 143.016,Z 519.344,A -85,B 0,C 180,E1 -24401.337,E2 -24401.337} C_VEL
LIN {X 0,Y 144.64,Z 516.5,A -85,B 0,C 180,E1 -24405.501,E2 -24405.501} C_VEL
LIN {X 0,Y 146.939,Z 512.631,A -85,B 0,C 180,E1 -24409.561,E2 -24409.561} C_VEL
LIN {X 0,Y 149.889,Z 507.633,A -85,B 0,C 180,E1 -24413.488,E2 -24413.488} C_VEL
LIN {X 0,Y 153.333,Z 501.336,A -85,B 0,C 180,E1 -24417.281,E2 -24417.281} C_VEL
LIN {X 0,Y 157.54,Z 493.44,A -85,B 0,C 180,E1 -24420.866,E2 -24420.866} C_VEL
LIN {X 0,Y 162.05,Z 483.627,A -85,B 0,C 180,E1 -24424.32,E2 -24424.32} C_VEL
LIN {X 0,Y 164.271,Z 477.92,A -85,B 0,C 180,E1 -24425.959,E2 -24425.959} C_VEL
LIN {X 0,Y 164.081,Z 470.377,A -85,B 0,C 180,E1 -24428.671,E2 -24428.671} C_VEL
LIN {X 0,Y 162.942,Z 461.548,A -85,B 0,C 180,E1 -24431.744,E2 -24431.744} C_VEL
LIN {X 0,Y 160.766,Z 453.563,A -85,B 0,C 180,E1 -24434.646,E2 -24434.646} C_VEL
LIN {X 0,Y 157.884,Z 446.701,A -85,B 0,C 180,E1 -24437.431,E2 -24437.431} C_VEL
LIN {X 0,Y 153.43,Z 438.585,A -85,B 0,C 180,E1 -24441.143,E2 -24441.143} C_VEL
LIN {X 0,Y 150.228,Z 433.219,A -85,B 0,C 180,E1 -24443.798,E2 -24443.798} C_VEL
LIN {X 0,Y 147.557,Z 429.644,A -85,B 0,C 180,E1 -24445.925,E2 -24445.925} C_VEL
LIN {X 0,Y 146.802,Z 427.992,A -85,B 0,C 180,E1 -24446.663,E2 -24446.663} C_VEL
LIN {X 0,Y 144.471,Z 425.941,A -85,B 0,C 180,E1 -24448.47,E2 -24448.47} C_VEL
LIN {X 0,Y 143.245,Z 423.317,A -85,B 0,C 180,E1 -24449.706,E2 -24449.706} C_VEL
LIN {X 0,Y 143.137,Z 422.653,A -85,B 0,C 180,E1 -24449.986,E2 -24449.986} C_VEL
LIN {X 0,Y 143.157,Z 422.654,A -85,B 0,C 180,E1 -24453.779,E2 -24453.779} C_VEL
LIN {X 0,Y 143.311,Z 422.632,A -85,B 0,C 180,E1 -24459.923,E2 -24459.923} C_VEL
LIN {X 0,Y 143.372,Z 422.624,A -85,B 0,C 180,E1 -24465.812,E2 -24465.812} C_VEL
LIN {X 0,Y 143.541,Z 422.604,A -85,B 0,C 180,E1 -24468.706,E2 -24468.706} C_VEL
LIN {X 0,Y 143.629,Z 422.594,A -85,B 0,C 180,E1 -24471.559,E2 -24471.559} C_VEL
LIN {X 0,Y 144.18,Z 422.531,A -85,B 0,C 180,E1 -24480,E2 -24480} C_VEL
LIN {X 0,Y 143.689,Z 422.589,A -85,B 0,C 180,E1 -24488.438,E2 -24488.438} C_VEL
LIN {X 0,Y 143.607,Z 422.843,A -85,B 0,C 180,E1 -24491.82,E2 -24491.82} C_VEL
LIN {X 0,Y 143.642,Z 424.401,A -85,B 0,C 180,E1 -24497.071,E2 -24497.071} C_VEL
LIN {X 0,Y 143.869,Z 426.064,A -85,B 0,C 180,E1 -24501.85,E2 -24501.85} C_VEL
LIN {X 0,Y 144.065,Z 427.714,A -85,B 0,C 180,E1 -24506.043,E2 -24506.043} C_VEL
LIN {X 0,Y 144.416,Z 430.006,A -85,B 0,C 180,E1 -24510.831,E2 -24510.831} C_VEL
LIN {X 0,Y 145.581,Z 433.065,A -85,B 0,C 180,E1 -24511.973,E2 -24511.973} C_VEL
LIN {X 0,Y 148.27,Z 436.574,A -85,B 0,C 180,E1 -24514.024,E2 -24514.024} C_VEL
LIN {X 0,Y 150.004,Z 440.361,A -85,B 0,C 180,E1 -24515.539,E2 -24515.539} C_VEL
LIN {X 0,Y 151.64,Z 442.815,A -85,B 0,C 180,E1 -24516.738,E2 -24516.738} C_VEL
LIN {X 0,Y 153.815,Z 447.142,A -85,B 0,C 180,E1 -24518.502,E2 -24518.502} C_VEL
LIN {X 0,Y 157.826,Z 456.368,A -85,B 0,C 180,E1 -24521.909,E2 -24521.909} C_VEL
LIN {X 0,Y 160.353,Z 464.332,A -85,B 0,C 180,E1 -24524.528,E2 -24524.528} C_VEL
LIN {X 0,Y 160.965,Z 474.261,A -85,B 0,C 180,E1 -24527.165,E2 -24527.165} C_VEL
LIN {X 0,Y 160.504,Z 485.152,A -85,B 0,C 180,E1 -24530.179,E2 -24530.179} C_VEL
LIN {X 0,Y 159.145,Z 495.388,A -85,B 0,C 180,E1 -24533.339,E2 -24533.339} C_VEL
LIN {X 0,Y 157.463,Z 503.189,A -85,B 0,C 180,E1 -24536.088,E2 -24536.088} C_VEL
LIN {X 0,Y 155.488,Z 508.119,A -85,B 0,C 180,E1 -24537.92,E2 -24537.92} C_VEL
LIN {X 0,Y 151.3,Z 516.429,A -85,B 0,C 180,E1 -24541.567,E2 -24541.567} C_VEL
LIN {X 0,Y 148.006,Z 523.155,A -85,B 0,C 180,E1 -24545.449,E2 -24545.449} C_VEL
LIN {X 0,Y 144.674,Z 529.303,A -85,B 0,C 180,E1 -24550.12,E2 -24550.12} C_VEL
LIN {X 0,Y 142.666,Z 533.316,A -85,B 0,C 180,E1 -24554.279,E2 -24554.279} C_VEL
LIN {X 0,Y 141.46,Z 536.302,A -85,B 0,C 180,E1 -24558.537,E2 -24558.537} C_VEL
LIN {X 0,Y 141.024,Z 537.731,A -85,B 0,C 180,E1 -24561.401,E2 -24561.401} C_VEL
LIN {X 0,Y 140.869,Z 539.227,A -85,B 0,C 180,E1 -24566.209,E2 -24566.209} C_VEL
LIN {X 0,Y 141.069,Z 539.623,A -85,B 0,C 180,E1 -24570,E2 -24570} C_VEL
LIN {X 0,Y 140.844,Z 539.241,A -85,B 0,C 180,E1 -24573.636,E2 -24573.636} C_VEL
LIN {X 0,Y 141.006,Z 537.702,A -85,B 0,C 180,E1 -24578.599,E2 -24578.599} C_VEL
LIN {X 0,Y 141.459,Z 536.262,A -85,B 0,C 180,E1 -24581.462,E2 -24581.462} C_VEL
LIN {X 0,Y 142.665,Z 533.259,A -85,B 0,C 180,E1 -24585.72,E2 -24585.72} C_VEL
LIN {X 0,Y 144.672,Z 529.223,A -85,B 0,C 180,E1 -24589.88,E2 -24589.88} C_VEL
LIN {X 0,Y 147.993,Z 523.043,A -85,B 0,C 180,E1 -24594.552,E2 -24594.552} C_VEL
LIN {X 0,Y 151.343,Z 516.295,A -85,B 0,C 180,E1 -24598.423,E2 -24598.423} C_VEL
LIN {X 0,Y 155.473,Z 507.952,A -85,B 0,C 180,E1 -24602.083,E2 -24602.083} C_VEL
LIN {X 0,Y 157.432,Z 502.987,A -85,B 0,C 180,E1 -24603.919,E2 -24603.919} C_VEL
LIN {X 0,Y 159.296,Z 494.122,A -85,B 0,C 180,E1 -24606.995,E2 -24606.995} C_VEL
LIN {X 0,Y 160.405,Z 484.843,A -85,B 0,C 180,E1 -24609.85,E2 -24609.85} C_VEL
LIN {X 0,Y 160.879,Z 475.286,A -85,B 0,C 180,E1 -24612.496,E2 -24612.496} C_VEL
LIN {X 0,Y 160.522,Z 465.907,A -85,B 0,C 180,E1 -24614.959,E2 -24614.959} C_VEL
LIN {X 0,Y 159.707,Z 461.949,A -85,B 0,C 180,E1 -24616.114,E2 -24616.114} C_VEL
LIN {X 0,Y 156.265,Z 452.729,A -85,B 0,C 180,E1 -24619.297,E2 -24619.297} C_VEL
LIN {X 0,Y 153.311,Z 446.403,A -85,B 0,C 180,E1 -24621.715,E2 -24621.715} C_VEL
LIN {X 0,Y 152.812,Z 445.559,A -85,B 0,C 180,E1 -24622.089,E2 -24622.089} C_VEL
LIN {X 0,Y 150.468,Z 442.458,A -85,B 0,C 180,E1 -24623.758,E2 -24623.758} C_VEL
LIN {X 0,Y 145.917,Z 438.812,A -85,B 0,C 180,E1 -24626.834,E2 -24626.834} C_VEL
LIN {X 0,Y 142.26,Z 436.351,A -85,B 0,C 180,E1 -24629.488,E2 -24629.488} C_VEL
LIN {X 0,Y 139.08,Z 433.378,A -85,B 0,C 180,E1 -24632.211,E2 -24632.211} C_VEL
LIN {X 0,Y 137.468,Z 430.176,A -85,B 0,C 180,E1 -24634.039,E2 -24634.039} C_VEL
LIN {X 0,Y 137.041,Z 428.832,A -85,B 0,C 180,E1 -24634.666,E2 -24634.666} C_VEL
LIN {X 0,Y 136.893,Z 427.258,A -85,B 0,C 180,E1 -24638.938,E2 -24638.938} C_VEL
LIN {X 0,Y 136.634,Z 425.351,A -85,B 0,C 180,E1 -24645.097,E2 -24645.097} C_VEL
LIN {X 0,Y 136.71,Z 424.501,A -85,B 0,C 180,E1 -24648.134,E2 -24648.134} C_VEL
LIN {X 0,Y 136.654,Z 423.784,A -85,B 0,C 180,E1 -24651.125,E2 -24651.125} C_VEL
LIN {X 0,Y 136.758,Z 423.449,A -85,B 0,C 180,E1 -24657.054,E2 -24657.054} C_VEL
LIN {X 0,Y 137.138,Z 423.402,A -85,B 0,C 180,E1 -24660,E2 -24660} C_VEL
LIN {X 0,Y 136.611,Z 423.469,A -85,B 0,C 180,E1 -24668.879,E2 -24668.879} C_VEL
LIN {X 0,Y 136.494,Z 423.482,A -85,B 0,C 180,E1 -24671.958,E2 -24671.958} C_VEL
LIN {X 0,Y 136.253,Z 423.511,A -85,B 0,C 180,E1 -24678.028,E2 -24678.028} C_VEL
LIN {X 0,Y 136.198,Z 423.517,A -85,B 0,C 180,E1 -24681.747,E2 -24681.747} C_VEL
LIN {X 0,Y 136.089,Z 423.664,A -85,B 0,C 180,E1 -24684.911,E2 -24684.911} C_VEL
LIN {X 0,Y 136.884,Z 425.981,A -85,B 0,C 180,E1 -24686.08,E2 -24686.08} C_VEL
LIN {X 0,Y 138.984,Z 428.388,A -85,B 0,C 180,E1 -24688.281,E2 -24688.281} C_VEL
LIN {X 0,Y 140.291,Z 429.396,A -85,B 0,C 180,E1 -24689.499,E2 -24689.499} C_VEL
LIN {X 0,Y 141.871,Z 432.455,A -85,B 0,C 180,E1 -24691.239,E2 -24691.239} C_VEL
LIN {X 0,Y 143.808,Z 434.563,A -85,B 0,C 180,E1 -24692.977,E2 -24692.977} C_VEL
LIN {X 0,Y 146.014,Z 438.185,A -85,B 0,C 180,E1 -24695.09,E2 -24695.09} C_VEL
LIN {X 0,Y 149.628,Z 444.493,A -85,B 0,C 180,E1 -24698.524,E2 -24698.524} C_VEL
LIN {X 0,Y 153.659,Z 452.483,A -85,B 0,C 180,E1 -24702.426,E2 -24702.426} C_VEL
LIN {X 0,Y 155.917,Z 459.117,A -85,B 0,C 180,E1 -24705.229,E2 -24705.229} C_VEL
LIN {X 0,Y 157.522,Z 467.29,A -85,B 0,C 180,E1 -24708.369,E2 -24708.369} C_VEL
LIN {X 0,Y 158.046,Z 475.624,A -85,B 0,C 180,E1 -24711.497,E2 -24711.497} C_VEL
LIN {X 0,Y 157.946,Z 479.738,A -85,B 0,C 180,E1 -24713.082,E2 -24713.082} C_VEL
LIN {X 0,Y 153.901,Z 488.845,A -85,B 0,C 180,E1 -24715.985,E2 -24715.985} C_VEL
LIN {X 0,Y 149.254,Z 497.71,A -85,B 0,C 180,E1 -24719.59,E2 -24719.59} C_VEL
LIN {X 0,Y 145.341,Z 504.829,A -85,B 0,C 180,E1 -24723.43,E2 -24723.43} C_VEL
LIN {X 0,Y 142.404,Z 509.63,A -85,B 0,C 180,E1 -24726.745,E2 -24726.745} C_VEL
LIN {X 0,Y 139.437,Z 514.293,A -85,B 0,C 180,E1 -24730.876,E2 -24730.876} C_VEL
LIN {X 0,Y 137.216,Z 517.849,A -85,B 0,C 180,E1 -24735.162,E2 -24735.162} C_VEL
LIN {X 0,Y 135.442,Z 520.794,A -85,B 0,C 180,E1 -24740.368,E2 -24740.368} C_VEL
LIN {X 0,Y 134.682,Z 522.033,A -85,B 0,C 180,E1 -24744.01,E2 -24744.01} C_VEL
LIN {X 0,Y 134.208,Z 522.858,A -85,B 0,C 180,E1 -24750,E2 -24750} C_VEL
LIN {X 0,Y 134.318,Z 522.662,A -85,B 0,C 180,E1 -24753,E2 -24753} C_VEL
LIN {X 0,Y 134.672,Z 522.08,A -85,B 0,C 180,E1 -24755.991,E2 -24755.991} C_VEL
LIN {X 0,Y 135.318,Z 520.993,A -85,B 0,C 180,E1 -24759.316,E2 -24759.316} C_VEL
LIN {X 0,Y 137.163,Z 517.976,A -85,B 0,C 180,E1 -24764.845,E2 -24764.845} C_VEL
LIN {X 0,Y 139.382,Z 514.466,A -85,B 0,C 180,E1 -24769.133,E2 -24769.133} C_VEL
LIN {X 0,Y 142.329,Z 509.85,A -85,B 0,C 180,E1 -24773.268,E2 -24773.268} C_VEL
LIN {X 0,Y 145.838,Z 503.996,A -85,B 0,C 180,E1 -24777.246,E2 -24777.246} C_VEL
LIN {X 0,Y 149.995,Z 496.687,A -85,B 0,C 180,E1 -24781.025,E2 -24781.025} C_VEL
LIN {X 0,Y 154.603,Z 487.708,A -85,B 0,C 180,E1 -24784.573,E2 -24784.573} C_VEL
LIN {X 0,Y 158.141,Z 479.208,A -85,B 0,C 180,E1 -24787.265,E2 -24787.265} C_VEL
LIN {X 0,Y 157.983,Z 471.02,A -85,B 0,C 180,E1 -24790.407,E2 -24790.407} C_VEL
LIN {X 0,Y 156.908,Z 462.969,A -85,B 0,C 180,E1 -24793.446,E2 -24793.446} C_VEL
LIN {X 0,Y 154.934,Z 455.858,A -85,B 0,C 180,E1 -24796.321,E2 -24796.321} C_VEL
LIN {X 0,Y 151.832,Z 448.707,A -85,B 0,C 180,E1 -24799.606,E2 -24799.606} C_VEL
LIN {X 0,Y 148.377,Z 442.192,A -85,B 0,C 180,E1 -24802.934,E2 -24802.934} C_VEL
LIN {X 0,Y 146.437,Z 438.601,A -85,B 0,C 180,E1 -24804.835,E2 -24804.835} C_VEL
LIN {X 0,Y 143.977,Z 434.984,A -85,B 0,C 180,E1 -24807.108,E2 -24807.108} C_VEL
LIN {X 0,Y 143.322,Z 433.89,A -85,B 0,C 180,E1 -24807.773,E2 -24807.773} C_VEL
LIN {X 0,Y 141.192,Z 431.462,A -85,B 0,C 180,E1 -24809.736,E2 -24809.736} C_VEL
LIN {X 0,Y 140.112,Z 429.062,A -85,B 0,C 180,E1 -24811.022,E2 -24811.022} C_VEL
LIN {X 0,Y 137.515,Z 426.954,A -85,B 0,C 180,E1 -24813.539,E2 -24813.539} C_VEL
LIN {X 0,Y 136.266,Z 424.515,A -85,B 0,C 180,E1 -24815.123,E2 -24815.123} C_VEL
LIN {X 0,Y 136.083,Z 423.532,A -85,B 0,C 180,E1 -24815.596,E2 -24815.596} C_VEL
LIN {X 0,Y 136.245,Z 423.514,A -85,B 0,C 180,E1 -24818.833,E2 -24818.833} C_VEL
LIN {X 0,Y 136.281,Z 423.51,A -85,B 0,C 180,E1 -24825.057,E2 -24825.057} C_VEL
LIN {X 0,Y 136.461,Z 423.488,A -85,B 0,C 180,E1 -24828.111,E2 -24828.111} C_VEL
LIN {X 0,Y 136.554,Z 423.477,A -85,B 0,C 180,E1 -24831.118,E2 -24831.118} C_VEL
LIN {X 0,Y 137.137,Z 423.408,A -85,B 0,C 180,E1 -24840,E2 -24840} C_VEL
LIN {X 0,Y 136.576,Z 423.476,A -85,B 0,C 180,E1 -24845.907,E2 -24845.907} C_VEL
LIN {X 0,Y 136.666,Z 423.836,A -85,B 0,C 180,E1 -24848.875,E2 -24848.875} C_VEL
LIN {X 0,Y 136.676,Z 424.694,A -85,B 0,C 180,E1 -24852.31,E2 -24852.31} C_VEL
LIN {X 0,Y 136.734,Z 426.34,A -85,B 0,C 180,E1 -24857.962,E2 -24857.962} C_VEL
LIN {X 0,Y 136.944,Z 427.882,A -85,B 0,C 180,E1 -24862.515,E2 -24862.515} C_VEL
LIN {X 0,Y 137.082,Z 429.082,A -85,B 0,C 180,E1 -24865.225,E2 -24865.225} C_VEL
LIN {X 0,Y 138.587,Z 432.621,A -85,B 0,C 180,E1 -24867.054,E2 -24867.054} C_VEL
LIN {X 0,Y 141.304,Z 435.948,A -85,B 0,C 180,E1 -24869.604,E2 -24869.604} C_VEL
LIN {X 0,Y 142.955,Z 439.711,A -85,B 0,C 180,E1 -24871.387,E2 -24871.387} C_VEL
LIN {X 0,Y 144.715,Z 442.208,A -85,B 0,C 180,E1 -24872.91,E2 -24872.91} C_VEL
LIN {X 0,Y 146.717,Z 446.471,A -85,B 0,C 180,E1 -24874.878,E2 -24874.878} C_VEL
LIN {X 0,Y 147.706,Z 448.213,A -85,B 0,C 180,E1 -24875.736,E2 -24875.736} C_VEL
LIN {X 0,Y 150.32,Z 454.213,A -85,B 0,C 180,E1 -24878.278,E2 -24878.278} C_VEL
LIN {X 0,Y 152.935,Z 460.733,A -85,B 0,C 180,E1 -24880.908,E2 -24880.908} C_VEL
LIN {X 0,Y 154.935,Z 467.886,A -85,B 0,C 180,E1 -24883.466,E2 -24883.466} C_VEL
LIN {X 0,Y 155.114,Z 477.51,A -85,B 0,C 180,E1 -24886.219,E2 -24886.219} C_VEL
LIN {X 0,Y 154.363,Z 487.177,A -85,B 0,C 180,E1 -24889.119,E2 -24889.119} C_VEL
LIN {X 0,Y 152.608,Z 497.808,A -85,B 0,C 180,E1 -24892.689,E2 -24892.689} C_VEL
LIN {X 0,Y 150.875,Z 504.444,A -85,B 0,C 180,E1 -24895.206,E2 -24895.206} C_VEL
LIN {X 0,Y 147.922,Z 510.679,A -85,B 0,C 180,E1 -24897.689,E2 -24897.689} C_VEL
LIN {X 0,Y 144.398,Z 517.241,A -85,B 0,C 180,E1 -24900.875,E2 -24900.875} C_VEL
LIN {X 0,Y 140.959,Z 523.722,A -85,B 0,C 180,E1 -24904.925,E2 -24904.925} C_VEL
LIN {X 0,Y 137.984,Z 528.869,A -85,B 0,C 180,E1 -24909.112,E2 -24909.112} C_VEL
LIN {X 0,Y 135.805,Z 532.882,A -85,B 0,C 180,E1 -24913.463,E2 -24913.463} C_VEL
LIN {X 0,Y 134.479,Z 535.868,A -85,B 0,C 180,E1 -24917.933,E2 -24917.933} C_VEL
LIN {X 0,Y 133.979,Z 537.297,A -85,B 0,C 180,E1 -24920.945,E2 -24920.945} C_VEL
LIN {X 0,Y 133.782,Z 538.877,A -85,B 0,C 180,E1 -24926.497,E2 -24926.497} C_VEL
LIN {X 0,Y 133.988,Z 539.192,A -85,B 0,C 180,E1 -24930,E2 -24930} C_VEL
LIN {X 0,Y 133.761,Z 538.889,A -85,B 0,C 180,E1 -24933.35,E2 -24933.35} C_VEL
LIN {X 0,Y 133.965,Z 537.268,A -85,B 0,C 180,E1 -24939.055,E2 -24939.055} C_VEL
LIN {X 0,Y 134.478,Z 535.827,A -85,B 0,C 180,E1 -24942.066,E2 -24942.066} C_VEL
LIN {X 0,Y 135.804,Z 532.823,A -85,B 0,C 180,E1 -24946.537,E2 -24946.537} C_VEL
LIN {X 0,Y 137.982,Z 528.787,A -85,B 0,C 180,E1 -24950.888,E2 -24950.888} C_VEL
LIN {X 0,Y 141.533,Z 522.607,A -85,B 0,C 180,E1 -24955.753,E2 -24955.753} C_VEL
LIN {X 0,Y 145.081,Z 515.857,A -85,B 0,C 180,E1 -24959.771,E2 -24959.771} C_VEL
LIN {X 0,Y 149.471,Z 507.514,A -85,B 0,C 180,E1 -24963.537,E2 -24963.537} C_VEL
LIN {X 0,Y 151.322,Z 502.531,A -85,B 0,C 180,E1 -24965.489,E2 -24965.489} C_VEL
LIN {X 0,Y 153.384,Z 493.243,A -85,B 0,C 180,E1 -24968.837,E2 -24968.837} C_VEL
LIN {X 0,Y 154.665,Z 483.038,A -85,B 0,C 180,E1 -24972.086,E2 -24972.086} C_VEL
LIN {X 0,Y 155.075,Z 472.655,A -85,B 0,C 180,E1 -24975.091,E2 -24975.091} C_VEL
LIN {X 0,Y 154.855,Z 467.438,A -85,B 0,C 180,E1 -24976.565,E2 -24976.565} C_VEL
LIN {X 0,Y 152.804,Z 460.607,A -85,B 0,C 180,E1 -24979.049,E2 -24979.049} C_VEL
LIN {X 0,Y 149.558,Z 452.247,A -85,B 0,C 180,E1 -24982.346,E2 -24982.346} C_VEL
LIN {X 0,Y 146.845,Z 446.676,A -85,B 0,C 180,E1 -24984.854,E2 -24984.854} C_VEL
LIN {X 0,Y 144.734,Z 442.297,A -85,B 0,C 180,E1 -24986.888,E2 -24986.888} C_VEL
LIN {X 0,Y 141.801,Z 437.534,A -85,B 0,C 180,E1 -24989.571,E2 -24989.571} C_VEL
LIN {X 0,Y 140.91,Z 435.427,A -85,B 0,C 180,E1 -24990.548,E2 -24990.548} C_VEL
LIN {X 0,Y 139.08,Z 433.378,A -85,B 0,C 180,E1 -24992.211,E2 -24992.211} C_VEL
LIN {X 0,Y 137.501,Z 432.232,A -85,B 0,C 180,E1 -24993.651,E2 -24993.651} C_VEL
LIN {X 0,Y 131.993,Z 431.792,A -85,B 0,C 180,E1 -24998.891,E2 -24998.891} C_VEL
LIN {X 0,Y 130.829,Z 430.658,A -85,B 0,C 180,E1 -25000.479,E2 -25000.479} C_VEL
LIN {X 0,Y 129.771,Z 427.718,A -85,B 0,C 180,E1 -25002.671,E2 -25002.671} C_VEL
LIN {X 0,Y 129.763,Z 426.393,A -85,B 0,C 180,E1 -25007.488,E2 -25007.488} C_VEL
LIN {X 0,Y 129.751,Z 425.631,A -85,B 0,C 180,E1 -25010.648,E2 -25010.648} C_VEL
LIN {X 0,Y 129.697,Z 424.42,A -85,B 0,C 180,E1 -25016.894,E2 -25016.894} C_VEL
LIN {X 0,Y 130.093,Z 424.28,A -85,B 0,C 180,E1 -25020,E2 -25020} C_VEL
LIN {X 0,Y 129.533,Z 424.348,A -85,B 0,C 180,E1 -25029.368,E2 -25029.368} C_VEL
LIN {X 0,Y 129.396,Z 424.364,A -85,B 0,C 180,E1 -25032.548,E2 -25032.548} C_VEL
LIN {X 0,Y 129.206,Z 424.545,A -85,B 0,C 180,E1 -25037.102,E2 -25037.102} C_VEL
LIN {X 0,Y 130.218,Z 427.315,A -85,B 0,C 180,E1 -25039.304,E2 -25039.304} C_VEL
LIN {X 0,Y 132.905,Z 429.863,A -85,B 0,C 180,E1 -25043.102,E2 -25043.102} C_VEL
LIN {X 0,Y 133.591,Z 430.423,A -85,B 0,C 180,E1 -25043.958,E2 -25043.958} C_VEL
LIN {X 0,Y 135.169,Z 433.531,A -85,B 0,C 180,E1 -25046.229,E2 -25046.229} C_VEL
LIN {X 0,Y 137.334,Z 435.828,A -85,B 0,C 180,E1 -25048.67,E2 -25048.67} C_VEL
LIN {X 0,Y 139.108,Z 438.974,A -85,B 0,C 180,E1 -25050.809,E2 -25050.809} C_VEL
LIN {X 0,Y 140.084,Z 440.011,A -85,B 0,C 180,E1 -25051.787,E2 -25051.787} C_VEL
LIN {X 0,Y 145.051,Z 448.952,A -85,B 0,C 180,E1 -25057.276,E2 -25057.276} C_VEL
LIN {X 0,Y 148.653,Z 456.837,A -85,B 0,C 180,E1 -25061.445,E2 -25061.445} C_VEL
LIN {X 0,Y 150.639,Z 463.322,A -85,B 0,C 180,E1 -25064.413,E2 -25064.413} C_VEL
LIN {X 0,Y 151.727,Z 470.173,A -85,B 0,C 180,E1 -25067.273,E2 -25067.273} C_VEL
LIN {X 0,Y 151.978,Z 478.16,A -85,B 0,C 180,E1 -25070.518,E2 -25070.518} C_VEL
LIN {X 0,Y 151.833,Z 481.269,A -85,B 0,C 180,E1 -25071.803,E2 -25071.803} C_VEL
LIN {X 0,Y 147.256,Z 490.891,A -85,B 0,C 180,E1 -25075.06,E2 -25075.06} C_VEL
LIN {X 0,Y 142.464,Z 499.462,A -85,B 0,C 180,E1 -25078.803,E2 -25078.803} C_VEL
LIN {X 0,Y 138.366,Z 506.282,A -85,B 0,C 180,E1 -25082.798,E2 -25082.798} C_VEL
LIN {X 0,Y 134.767,Z 511.745,A -85,B 0,C 180,E1 -25086.976,E2 -25086.976} C_VEL
LIN {X 0,Y 131.894,Z 516.022,A -85,B 0,C 180,E1 -25091.355,E2 -25091.355} C_VEL
LIN {X 0,Y 130.384,Z 518.281,A -85,B 0,C 180,E1 -25094.365,E2 -25094.365} C_VEL
LIN {X 0,Y 128.382,Z 521.363,A -85,B 0,C 180,E1 -25100.191,E2 -25100.191} C_VEL
LIN {X 0,Y 127.647,Z 522.465,A -85,B 0,C 180,E1 -25103.678,E2 -25103.678} C_VEL
LIN {X 0,Y 127.13,Z 523.289,A -85,B 0,C 180,E1 -25110,E2 -25110} C_VEL
LIN {X 0,Y 127.251,Z 523.093,A -85,B 0,C 180,E1 -25113.166,E2 -25113.166} C_VEL
LIN {X 0,Y 127.636,Z 522.51,A -85,B 0,C 180,E1 -25116.323,E2 -25116.323} C_VEL
LIN {X 0,Y 129.157,Z 520.206,A -85,B 0,C 180,E1 -25122.572,E2 -25122.572} C_VEL
LIN {X 0,Y 131.04,Z 517.361,A -85,B 0,C 180,E1 -25127.157,E2 -25127.157} C_VEL
LIN {X 0,Y 133.674,Z 513.491,A -85,B 0,C 180,E1 -25131.595,E2 -25131.595} C_VEL
LIN {X 0,Y 136.998,Z 508.493,A -85,B 0,C 180,E1 -25135.853,E2 -25135.853} C_VEL
LIN {X 0,Y 140.889,Z 502.195,A -85,B 0,C 180,E1 -25139.923,E2 -25139.923} C_VEL
LIN {X 0,Y 145.571,Z 494.296,A -85,B 0,C 180,E1 -25143.725,E2 -25143.725} C_VEL
LIN {X 0,Y 150.055,Z 485.521,A -85,B 0,C 180,E1 -25147.015,E2 -25147.015} C_VEL
LIN {X 0,Y 152.045,Z 480.656,A -85,B 0,C 180,E1 -25148.609,E2 -25148.609} C_VEL
LIN {X 0,Y 151.969,Z 471.746,A -85,B 0,C 180,E1 -25152.273,E2 -25152.273} C_VEL
LIN {X 0,Y 151.154,Z 465.512,A -85,B 0,C 180,E1 -25154.841,E2 -25154.841} C_VEL
LIN {X 0,Y 149.845,Z 460.279,A -85,B 0,C 180,E1 -25157.15,E2 -25157.15} C_VEL
LIN {X 0,Y 147.305,Z 453.754,A -85,B 0,C 180,E1 -25160.393,E2 -25160.393} C_VEL
LIN {X 0,Y 143.961,Z 447.031,A -85,B 0,C 180,E1 -25164.138,E2 -25164.138} C_VEL
LIN {X 0,Y 141.484,Z 442.622,A -85,B 0,C 180,E1 -25166.879,E2 -25166.879} C_VEL
LIN {X 0,Y 140.059,Z 439.967,A -85,B 0,C 180,E1 -25168.545,E2 -25168.545} C_VEL
LIN {X 0,Y 138.996,Z 438.816,A -85,B 0,C 180,E1 -25169.627,E2 -25169.627} C_VEL
LIN {X 0,Y 136.997,Z 435.254,A -85,B 0,C 180,E1 -25172.088,E2 -25172.088} C_VEL
LIN {X 0,Y 134.715,Z 432.859,A -85,B 0,C 180,E1 -25174.714,E2 -25174.714} C_VEL
LIN {X 0,Y 133.395,Z 430.091,A -85,B 0,C 180,E1 -25176.725,E2 -25176.725} C_VEL
LIN {X 0,Y 130.476,Z 427.704,A -85,B 0,C 180,E1 -25180.736,E2 -25180.736} C_VEL
LIN {X 0,Y 129.277,Z 424.936,A -85,B 0,C 180,E1 -25183.213,E2 -25183.213} C_VEL
LIN {X 0,Y 129.199,Z 424.388,A -85,B 0,C 180,E1 -25183.609,E2 -25183.609} C_VEL
LIN {X 0,Y 129.402,Z 424.367,A -85,B 0,C 180,E1 -25187.855,E2 -25187.855} C_VEL
LIN {X 0,Y 129.482,Z 424.357,A -85,B 0,C 180,E1 -25190.628,E2 -25190.628} C_VEL
LIN {X 0,Y 130.092,Z 424.286,A -85,B 0,C 180,E1 -25200,E2 -25200} C_VEL
LIN {X 0,Y 129.65,Z 425.063,A -85,B 0,C 180,E1 -25206.224,E2 -25206.224} C_VEL
LIN {X 0,Y 129.76,Z 425.678,A -85,B 0,C 180,E1 -25209.351,E2 -25209.351} C_VEL
LIN {X 0,Y 129.747,Z 426.527,A -85,B 0,C 180,E1 -25212.835,E2 -25212.835} C_VEL
LIN {X 0,Y 129.828,Z 427.932,A -85,B 0,C 180,E1 -25217.22,E2 -25217.22} C_VEL
LIN {X 0,Y 131.073,Z 431.127,A -85,B 0,C 180,E1 -25219.58,E2 -25219.58} C_VEL
LIN {X 0,Y 134.472,Z 435.35,A -85,B 0,C 180,E1 -25224.051,E2 -25224.051} C_VEL
LIN {X 0,Y 136.183,Z 439.257,A -85,B 0,C 180,E1 -25226.43,E2 -25226.43} C_VEL
LIN {X 0,Y 138.098,Z 441.917,A -85,B 0,C 180,E1 -25228.497,E2 -25228.497} C_VEL
LIN {X 0,Y 139.973,Z 446.047,A -85,B 0,C 180,E1 -25230.765,E2 -25230.765} C_VEL
LIN {X 0,Y 140.837,Z 447.279,A -85,B 0,C 180,E1 -25231.6,E2 -25231.6} C_VEL
LIN {X 0,Y 142.584,Z 451.48,A -85,B 0,C 180,E1 -25233.677,E2 -25233.677} C_VEL
LIN {X 0,Y 143.843,Z 454.169,A -85,B 0,C 180,E1 -25235.036,E2 -25235.036} C_VEL
LIN {X 0,Y 146.82,Z 461.684,A -85,B 0,C 180,E1 -25238.483,E2 -25238.483} C_VEL
LIN {X 0,Y 148.924,Z 468.715,A -85,B 0,C 180,E1 -25241.352,E2 -25241.352} C_VEL
LIN {X 0,Y 149.511,Z 472.924,A -85,B 0,C 180,E1 -25242.838,E2 -25242.838} C_VEL
LIN {X 0,Y 149.048,Z 482.856,A -85,B 0,C 180,E1 -25245.922,E2 -25245.922} C_VEL
LIN {X 0,Y 147.813,Z 491.701,A -85,B 0,C 180,E1 -25248.853,E2 -25248.853} C_VEL
LIN {X 0,Y 145.895,Z 500.468,A -85,B 0,C 180,E1 -25252.107,E2 -25252.107} C_VEL
LIN {X 0,Y 144.312,Z 505.66,A -85,B 0,C 180,E1 -25254.239,E2 -25254.239} C_VEL
LIN {X 0,Y 140.359,Z 512.993,A -85,B 0,C 180,E1 -25257.434,E2 -25257.434} C_VEL
LIN {X 0,Y 136.094,Z 520.385,A -85,B 0,C 180,E1 -25261.593,E2 -25261.593} C_VEL
LIN {X 0,Y 133.332,Z 525.121,A -85,B 0,C 180,E1 -25265.058,E2 -25265.058} C_VEL
LIN {X 0,Y 130.468,Z 529.885,A -85,B 0,C 180,E1 -25269.504,E2 -25269.504} C_VEL
LIN {X 0,Y 128.409,Z 533.54,A -85,B 0,C 180,E1 -25274.118,E2 -25274.118} C_VEL
LIN {X 0,Y 127.511,Z 535.434,A -85,B 0,C 180,E1 -25277.263,E2 -25277.263} C_VEL
LIN {X 0,Y 126.699,Z 537.893,A -85,B 0,C 180,E1 -25283.63,E2 -25283.63} C_VEL
LIN {X 0,Y 126.699,Z 538.528,A -85,B 0,C 180,E1 -25286.82,E2 -25286.82} C_VEL
LIN {X 0,Y 126.907,Z 538.761,A -85,B 0,C 180,E1 -25290,E2 -25290} C_VEL
LIN {X 0,Y 126.699,Z 538.515,A -85,B 0,C 180,E1 -25293.18,E2 -25293.18} C_VEL
LIN {X 0,Y 126.695,Z 537.871,A -85,B 0,C 180,E1 -25296.369,E2 -25296.369} C_VEL
LIN {X 0,Y 126.93,Z 536.833,A -85,B 0,C 180,E1 -25299.561,E2 -25299.561} C_VEL
LIN {X 0,Y 127.496,Z 535.391,A -85,B 0,C 180,E1 -25302.738,E2 -25302.738} C_VEL
LIN {X 0,Y 128.958,Z 532.386,A -85,B 0,C 180,E1 -25307.442,E2 -25307.442} C_VEL
LIN {X 0,Y 131.344,Z 528.351,A -85,B 0,C 180,E1 -25311.997,E2 -25311.997} C_VEL
LIN {X 0,Y 135.11,Z 522.168,A -85,B 0,C 180,E1 -25317.074,E2 -25317.074} C_VEL
LIN {X 0,Y 138.893,Z 515.418,A -85,B 0,C 180,E1 -25321.242,E2 -25321.242} C_VEL
LIN {X 0,Y 143.565,Z 507.076,A -85,B 0,C 180,E1 -25325.114,E2 -25325.114} C_VEL
LIN {X 0,Y 145.353,Z 502.077,A -85,B 0,C 180,E1 -25327.185,E2 -25327.185} C_VEL
LIN {X 0,Y 147.506,Z 492.913,A -85,B 0,C 180,E1 -25330.643,E2 -25330.643} C_VEL
LIN {X 0,Y 148.933,Z 482.743,A -85,B 0,C 180,E1 -25334.044,E2 -25334.044} C_VEL
LIN {X 0,Y 149.461,Z 472.518,A -85,B 0,C 180,E1 -25337.183,E2 -25337.183} C_VEL
LIN {X 0,Y 148.866,Z 468.415,A -85,B 0,C 180,E1 -25338.628,E2 -25338.628} C_VEL
LIN {X 0,Y 145.983,Z 459.683,A -85,B 0,C 180,E1 -25342.31,E2 -25342.31} C_VEL
LIN {X 0,Y 143.13,Z 452.419,A -85,B 0,C 180,E1 -25345.62,E2 -25345.62} C_VEL
LIN {X 0,Y 140.228,Z 446.498,A -85,B 0,C 180,E1 -25348.773,E2 -25348.773} C_VEL
LIN {X 0,Y 138.201,Z 442.341,A -85,B 0,C 180,E1 -25351.111,E2 -25351.111} C_VEL
LIN {X 0,Y 137.617,Z 441.166,A -85,B 0,C 180,E1 -25351.81,E2 -25351.81} C_VEL
LIN {X 0,Y 135.302,Z 437.651,A -85,B 0,C 180,E1 -25354.42,E2 -25354.42} C_VEL
LIN {X 0,Y 134.295,Z 434.994,A -85,B 0,C 180,E1 -25355.918,E2 -25355.918} C_VEL
LIN {X 0,Y 130.993,Z 430.993,A -85,B 0,C 180,E1 -25360.204,E2 -25360.204} C_VEL
LIN {X 0,Y 130.829,Z 430.658,A -85,B 0,C 180,E1 -25360.479,E2 -25360.479} C_VEL
LIN {X 0,Y 129.732,Z 429.737,A -85,B 0,C 180,E1 -25362.082,E2 -25362.082} C_VEL
LIN {X 0,Y 127.634,Z 430.432,A -85,B 0,C 180,E1 -25364.896,E2 -25364.896} C_VEL
LIN {X 0,Y 125.747,Z 431.535,A -85,B 0,C 180,E1 -25367.848,E2 -25367.848} C_VEL
LIN {X 0,Y 124.977,Z 431.182,A -85,B 0,C 180,E1 -25369.662,E2 -25369.662} C_VEL
LIN {X 0,Y 123.492,Z 427.63,A -85,B 0,C 180,E1 -25377.962,E2 -25377.962} C_VEL
LIN {X 0,Y 123.494,Z 426.935,A -85,B 0,C 180,E1 -25380,E2 -25380} C_VEL
LIN {X 0,Y 127.211,Z 431.37,A -85,B 0,C 180,E1 -25396.242,E2 -25396.242} C_VEL
LIN {X 0,Y 128.225,Z 434.092,A -85,B 0,C 180,E1 -25398.785,E2 -25398.785} C_VEL
LIN {X 0,Y 130.958,Z 436.887,A -85,B 0,C 180,E1 -25403.106,E2 -25403.106} C_VEL
LIN {X 0,Y 132.417,Z 439.854,A -85,B 0,C 180,E1 -25405.542,E2 -25405.542} C_VEL
LIN {X 0,Y 134.314,Z 442.398,A -85,B 0,C 180,E1 -25408.095,E2 -25408.095} C_VEL
LIN {X 0,Y 135.351,Z 444.377,A -85,B 0,C 180,E1 -25409.557,E2 -25409.557} C_VEL
LIN {X 0,Y 136.813,Z 446.53,A -85,B 0,C 180,E1 -25411.384,E2 -25411.384} C_VEL
LIN {X 0,Y 140.408,Z 453.498,A -85,B 0,C 180,E1 -25416.025,E2 -25416.025} C_VEL
LIN {X 0,Y 143.793,Z 461.659,A -85,B 0,C 180,E1 -25420.724,E2 -25420.724} C_VEL
LIN {X 0,Y 145.242,Z 467.205,A -85,B 0,C 180,E1 -25423.463,E2 -25423.463} C_VEL
LIN {X 0,Y 146.027,Z 474.595,A -85,B 0,C 180,E1 -25426.796,E2 -25426.796} C_VEL
LIN {X 0,Y 145.832,Z 482.559,A -85,B 0,C 180,E1 -25430.318,E2 -25430.318} C_VEL
LIN {X 0,Y 141.511,Z 491.325,A -85,B 0,C 180,E1 -25433.418,E2 -25433.418} C_VEL
LIN {X 0,Y 136.441,Z 499.896,A -85,B 0,C 180,E1 -25437.259,E2 -25437.259} C_VEL
LIN {X 0,Y 132.099,Z 506.716,A -85,B 0,C 180,E1 -25441.392,E2 -25441.392} C_VEL
LIN {X 0,Y 128.268,Z 512.178,A -85,B 0,C 180,E1 -25445.737,E2 -25445.737} C_VEL
LIN {X 0,Y 125.187,Z 516.456,A -85,B 0,C 180,E1 -25450.316,E2 -25450.316} C_VEL
LIN {X 0,Y 123.574,Z 518.714,A -85,B 0,C 180,E1 -25453.479,E2 -25453.479} C_VEL
LIN {X 0,Y 122.307,Z 520.544,A -85,B 0,C 180,E1 -25456.712,E2 -25456.712} C_VEL
LIN {X 0,Y 121.323,Z 521.918,A -85,B 0,C 180,E1 -25459.992,E2 -25459.992} C_VEL
LIN {X 0,Y 120.19,Z 523.496,A -85,B 0,C 180,E1 -25466.648,E2 -25466.648} C_VEL
LIN {X 0,Y 120.054,Z 523.72,A -85,B 0,C 180,E1 -25470,E2 -25470} C_VEL
LIN {X 0,Y 120.186,Z 523.524,A -85,B 0,C 180,E1 -25473.353,E2 -25473.353} C_VEL
LIN {X 0,Y 121.195,Z 522.1,A -85,B 0,C 180,E1 -25479.659,E2 -25479.659} C_VEL
LIN {X 0,Y 122.253,Z 520.637,A -85,B 0,C 180,E1 -25483.295,E2 -25483.295} C_VEL
LIN {X 0,Y 124.274,Z 517.792,A -85,B 0,C 180,E1 -25488.122,E2 -25488.122} C_VEL
LIN {X 0,Y 127.119,Z 513.921,A -85,B 0,C 180,E1 -25492.769,E2 -25492.769} C_VEL
LIN {X 0,Y 130.66,Z 508.923,A -85,B 0,C 180,E1 -25497.207,E2 -25497.207} C_VEL
LIN {X 0,Y 134.799,Z 502.624,A -85,B 0,C 180,E1 -25501.425,E2 -25501.425} C_VEL
LIN {X 0,Y 139.739,Z 494.725,A -85,B 0,C 180,E1 -25505.337,E2 -25505.337} C_VEL
LIN {X 0,Y 144.307,Z 486.267,A -85,B 0,C 180,E1 -25508.595,E2 -25508.595} C_VEL
LIN {X 0,Y 145.752,Z 483.195,A -85,B 0,C 180,E1 -25509.62,E2 -25509.62} C_VEL
LIN {X 0,Y 146.1,Z 480.144,A -85,B 0,C 180,E1 -25510.951,E2 -25510.951} C_VEL
LIN {X 0,Y 146.051,Z 472.542,A -85,B 0,C 180,E1 -25514.292,E2 -25514.292} C_VEL
LIN {X 0,Y 145.063,Z 466.028,A -85,B 0,C 180,E1 -25517.291,E2 -25517.291} C_VEL
LIN {X 0,Y 143.204,Z 460.166,A -85,B 0,C 180,E1 -25520.357,E2 -25520.357} C_VEL
LIN {X 0,Y 139.998,Z 452.757,A -85,B 0,C 180,E1 -25524.738,E2 -25524.738} C_VEL
LIN {X 0,Y 136.734,Z 446.279,A -85,B 0,C 180,E1 -25529.07,E2 -25529.07} C_VEL
LIN {X 0,Y 133.187,Z 440.815,A -85,B 0,C 180,E1 -25533.775,E2 -25533.775} C_VEL
LIN {X 0,Y 131.096,Z 437.287,A -85,B 0,C 180,E1 -25537.024,E2 -25537.024} C_VEL
LIN {X 0,Y 130.874,Z 436.591,A -85,B 0,C 180,E1 -25537.504,E2 -25537.504} C_VEL
LIN {X 0,Y 128.371,Z 434.299,A -85,B 0,C 180,E1 -25541.444,E2 -25541.444} C_VEL
LIN {X 0,Y 127.212,Z 431.3,A -85,B 0,C 180,E1 -25544.376,E2 -25544.376} C_VEL
LIN {X 0,Y 123.707,Z 427.445,A -85,B 0,C 180,E1 -25560,E2 -25560} C_VEL
LIN {X 0,Y 124.582,Z 430.394,A -85,B 0,C 180,E1 -25568.107,E2 -25568.107} C_VEL
LIN {X 0,Y 127.797,Z 434.453,A -85,B 0,C 180,E1 -25576.165,E2 -25576.165} C_VEL
LIN {X 0,Y 129.09,Z 437.916,A -85,B 0,C 180,E1 -25579.066,E2 -25579.066} C_VEL
LIN {X 0,Y 131.721,Z 441.687,A -85,B 0,C 180,E1 -25583.068,E2 -25583.068} C_VEL
LIN {X 0,Y 133.409,Z 445.672,A -85,B 0,C 180,E1 -25585.761,E2 -25585.761} C_VEL
LIN {X 0,Y 135.017,Z 448.673,A -85,B 0,C 180,E1 -25587.935,E2 -25587.935} C_VEL
LIN {X 0,Y 137.631,Z 454.599,A -85,B 0,C 180,E1 -25591.49,E2 -25591.49} C_VEL
LIN {X 0,Y 140.368,Z 461.421,A -85,B 0,C 180,E1 -25595.155,E2 -25595.155} C_VEL
LIN {X 0,Y 142.732,Z 468.799,A -85,B 0,C 180,E1 -25598.648,E2 -25598.648} C_VEL
LIN {X 0,Y 143.97,Z 474.705,A -85,B 0,C 180,E1 -25601.151,E2 -25601.151} C_VEL
LIN {X 0,Y 143.312,Z 484.009,A -85,B 0,C 180,E1 -25604.275,E2 -25604.275} C_VEL
LIN {X 0,Y 141.651,Z 493.666,A -85,B 0,C 180,E1 -25607.709,E2 -25607.709} C_VEL
LIN {X 0,Y 139.01,Z 503.551,A -85,B 0,C 180,E1 -25611.732,E2 -25611.732} C_VEL
LIN {X 0,Y 136.929,Z 508.32,A -85,B 0,C 180,E1 -25613.825,E2 -25613.825} C_VEL
LIN {X 0,Y 132.074,Z 516.373,A -85,B 0,C 180,E1 -25617.85,E2 -25617.85} C_VEL
LIN {X 0,Y 128.183,Z 522.857,A -85,B 0,C 180,E1 -25622.222,E2 -25622.222} C_VEL
LIN {X 0,Y 124.764,Z 528.003,A -85,B 0,C 180,E1 -25626.776,E2 -25626.776} C_VEL
LIN {X 0,Y 122.162,Z 532.013,A -85,B 0,C 180,E1 -25631.553,E2 -25631.553} C_VEL
LIN {X 0,Y 120.556,Z 535,A -85,B 0,C 180,E1 -25636.515,E2 -25636.515} C_VEL
LIN {X 0,Y 119.637,Z 537.46,A -85,B 0,C 180,E1 -25643.252,E2 -25643.252} C_VEL
LIN {X 0,Y 119.616,Z 538.179,A -85,B 0,C 180,E1 -25647.228,E2 -25647.228} C_VEL
LIN {X 0,Y 119.809,Z 538.328,A -85,B 0,C 180,E1 -25650,E2 -25650} C_VEL
LIN {X 0,Y 119.602,Z 538.082,A -85,B 0,C 180,E1 -25653.368,E2 -25653.368} C_VEL
LIN {X 0,Y 119.634,Z 537.438,A -85,B 0,C 180,E1 -25656.747,E2 -25656.747} C_VEL
LIN {X 0,Y 119.918,Z 536.399,A -85,B 0,C 180,E1 -25660.126,E2 -25660.126} C_VEL
LIN {X 0,Y 120.544,Z 534.956,A -85,B 0,C 180,E1 -25663.486,E2 -25663.486} C_VEL
LIN {X 0,Y 122.161,Z 531.95,A -85,B 0,C 180,E1 -25668.446,E2 -25668.446} C_VEL
LIN {X 0,Y 124.761,Z 527.916,A -85,B 0,C 180,E1 -25673.223,E2 -25673.223} C_VEL
LIN {X 0,Y 128.755,Z 521.729,A -85,B 0,C 180,E1 -25678.529,E2 -25678.529} C_VEL
LIN {X 0,Y 132.822,Z 514.979,A -85,B 0,C 180,E1 -25682.844,E2 -25682.844} C_VEL
LIN {X 0,Y 137.729,Z 506.635,A -85,B 0,C 180,E1 -25686.839,E2 -25686.839} C_VEL
LIN {X 0,Y 139.995,Z 499.791,A -85,B 0,C 180,E1 -25689.797,E2 -25689.797} C_VEL
LIN {X 0,Y 141.964,Z 491.324,A -85,B 0,C 180,E1 -25693.082,E2 -25693.082} C_VEL
LIN {X 0,Y 143.402,Z 482.261,A -85,B 0,C 180,E1 -25696.222,E2 -25696.222} C_VEL
LIN {X 0,Y 143.883,Z 474.138,A -85,B 0,C 180,E1 -25698.941,E2 -25698.941} C_VEL
LIN {X 0,Y 142.234,Z 467.464,A -85,B 0,C 180,E1 -25701.857,E2 -25701.857} C_VEL
LIN {X 0,Y 140.224,Z 461.27,A -85,B 0,C 180,E1 -25704.804,E2 -25704.804} C_VEL
LIN {X 0,Y 138.491,Z 456.726,A -85,B 0,C 180,E1 -25707.161,E2 -25707.161} C_VEL
LIN {X 0,Y 137.087,Z 452.973,A -85,B 0,C 180,E1 -25709.158,E2 -25709.158} C_VEL
LIN {X 0,Y 134.875,Z 448.379,A -85,B 0,C 180,E1 -25712.033,E2 -25712.033} C_VEL
LIN {X 0,Y 134.536,Z 447.248,A -85,B 0,C 180,E1 -25712.631,E2 -25712.631} C_VEL
LIN {X 0,Y 132.29,Z 443.481,A -85,B 0,C 180,E1 -25715.582,E2 -25715.582} C_VEL
LIN {X 0,Y 131.38,Z 441.031,A -85,B 0,C 180,E1 -25717.181,E2 -25717.181} C_VEL
LIN {X 0,Y 128.546,Z 436.886,A -85,B 0,C 180,E1 -25721.574,E2 -25721.574} C_VEL
LIN {X 0,Y 127.689,Z 434.298,A -85,B 0,C 180,E1 -25723.616,E2 -25723.616} C_VEL
LIN {X 0,Y 124.977,Z 431.182,A -85,B 0,C 180,E1 -25729.662,E2 -25729.662} C_VEL
LIN {X 0,Y 124.137,Z 430.442,A -85,B 0,C 180,E1 -25732.333,E2 -25732.333} C_VEL
LIN {X 0,Y 123.334,Z 430.88,A -85,B 0,C 180,E1 -25735.058,E2 -25735.058} C_VEL
LIN {X 0,Y 122.007,Z 435.002,A -85,B 0,C 180,E1 -25744.328,E2 -25744.328} C_VEL
LIN {X 0,Y 124.971,Z 438.087,A -85,B 0,C 180,E1 -25755.494,E2 -25755.494} C_VEL
LIN {X 0,Y 126.461,Z 441.532,A -85,B 0,C 180,E1 -25759.478,E2 -25759.478} C_VEL
LIN {X 0,Y 128.194,Z 443.599,A -85,B 0,C 180,E1 -25762.567,E2 -25762.567} C_VEL
LIN {X 0,Y 129.878,Z 446.741,A -85,B 0,C 180,E1 -25765.652,E2 -25765.652} C_VEL
LIN {X 0,Y 132.798,Z 451.677,A -85,B 0,C 180,E1 -25770.183,E2 -25770.183} C_VEL
LIN {X 0,Y 136.175,Z 459.143,A -85,B 0,C 180,E1 -25775.494,E2 -25775.494} C_VEL
LIN {X 0,Y 138.462,Z 465.35,A -85,B 0,C 180,E1 -25779.383,E2 -25779.383} C_VEL
LIN {X 0,Y 139.593,Z 469.764,A -85,B 0,C 180,E1 -25781.843,E2 -25781.843} C_VEL
LIN {X 0,Y 140.165,Z 475.283,A -85,B 0,C 180,E1 -25784.586,E2 -25784.586} C_VEL
LIN {X 0,Y 139.939,Z 483.036,A -85,B 0,C 180,E1 -25788.286,E2 -25788.286} C_VEL
LIN {X 0,Y 139.6,Z 484.915,A -85,B 0,C 180,E1 -25789.12,E2 -25789.12} C_VEL
LIN {X 0,Y 135.011,Z 493.34,A -85,B 0,C 180,E1 -25792.292,E2 -25792.292} C_VEL
LIN {X 0,Y 129.738,Z 501.548,A -85,B 0,C 180,E1 -25796.272,E2 -25796.272} C_VEL
LIN {X 0,Y 125.92,Z 507.149,A -85,B 0,C 180,E1 -25799.847,E2 -25799.847} C_VEL
LIN {X 0,Y 121.84,Z 512.611,A -85,B 0,C 180,E1 -25804.366,E2 -25804.366} C_VEL
LIN {X 0,Y 118.538,Z 516.888,A -85,B 0,C 180,E1 -25809.162,E2 -25809.162} C_VEL
LIN {X 0,Y 116.787,Z 519.147,A -85,B 0,C 180,E1 -25812.489,E2 -25812.489} C_VEL
LIN {X 0,Y 115.425,Z 520.976,A -85,B 0,C 180,E1 -25815.904,E2 -25815.904} C_VEL
LIN {X 0,Y 114.272,Z 522.467,A -85,B 0,C 180,E1 -25819.751,E2 -25819.751} C_VEL
LIN {X 0,Y 113.129,Z 523.927,A -85,B 0,C 180,E1 -25826.439,E2 -25826.439} C_VEL
LIN {X 0,Y 112.979,Z 524.151,A -85,B 0,C 180,E1 -25830,E2 -25830} C_VEL
LIN {X 0,Y 113.125,Z 523.954,A -85,B 0,C 180,E1 -25833.562,E2 -25833.562} C_VEL
LIN {X 0,Y 114.322,Z 522.413,A -85,B 0,C 180,E1 -25840.628,E2 -25840.628} C_VEL
LIN {X 0,Y 115.356,Z 521.068,A -85,B 0,C 180,E1 -25844.105,E2 -25844.105} C_VEL
LIN {X 0,Y 117.554,Z 518.223,A -85,B 0,C 180,E1 -25849.198,E2 -25849.198} C_VEL
LIN {X 0,Y 120.627,Z 514.351,A -85,B 0,C 180,E1 -25854.07,E2 -25854.07} C_VEL
LIN {X 0,Y 124.404,Z 509.353,A -85,B 0,C 180,E1 -25858.699,E2 -25858.699} C_VEL
LIN {X 0,Y 128.814,Z 503.053,A -85,B 0,C 180,E1 -25863.066,E2 -25863.066} C_VEL
LIN {X 0,Y 134.03,Z 495.153,A -85,B 0,C 180,E1 -25867.087,E2 -25867.087} C_VEL
LIN {X 0,Y 138.592,Z 487.149,A -85,B 0,C 180,E1 -25870.262,E2 -25870.262} C_VEL
LIN {X 0,Y 139.503,Z 485.345,A -85,B 0,C 180,E1 -25870.915,E2 -25870.915} C_VEL
LIN {X 0,Y 140.04,Z 483.462,A -85,B 0,C 180,E1 -25871.68,E2 -25871.68} C_VEL
LIN {X 0,Y 140.312,Z 475.53,A -85,B 0,C 180,E1 -25875.473,E2 -25875.473} C_VEL
LIN {X 0,Y 139.716,Z 470.088,A -85,B 0,C 180,E1 -25878.202,E2 -25878.202} C_VEL
LIN {X 0,Y 137.708,Z 463.128,A -85,B 0,C 180,E1 -25882.234,E2 -25882.234} C_VEL
LIN {X 0,Y 135.839,Z 458.358,A -85,B 0,C 180,E1 -25885.311,E2 -25885.311} C_VEL
LIN {X 0,Y 132.985,Z 452.02,A -85,B 0,C 180,E1 -25889.864,E2 -25889.864} C_VEL
LIN {X 0,Y 130.093,Z 447.052,A -85,B 0,C 180,E1 -25894.394,E2 -25894.394} C_VEL
LIN {X 0,Y 127.589,Z 442.63,A -85,B 0,C 180,E1 -25899.02,E2 -25899.02} C_VEL
LIN {X 0,Y 125.963,Z 440.803,A -85,B 0,C 180,E1 -25902.129,E2 -25902.129} C_VEL
LIN {X 0,Y 124.931,Z 437.873,A -85,B 0,C 180,E1 -25905.336,E2 -25905.336} C_VEL
LIN {X 0,Y 122.236,Z 434.472,A -85,B 0,C 180,E1 -25920,E2 -25920} C_VEL
LIN {X 0,Y 123.239,Z 437.79,A -85,B 0,C 180,E1 -25929.023,E2 -25929.023} C_VEL
LIN {X 0,Y 125.47,Z 440.995,A -85,B 0,C 180,E1 -25935.222,E2 -25935.222} C_VEL
LIN {X 0,Y 126.759,Z 444.645,A -85,B 0,C 180,E1 -25938.59,E2 -25938.59} C_VEL
LIN {X 0,Y 128.386,Z 447.13,A -85,B 0,C 180,E1 -25941.469,E2 -25941.469} C_VEL
LIN {X 0,Y 131.113,Z 453.402,A -85,B 0,C 180,E1 -25946.333,E2 -25946.333} C_VEL
LIN {X 0,Y 133.328,Z 459.129,A -85,B 0,C 180,E1 -25950.051,E2 -25950.051} C_VEL
LIN {X 0,Y 135.701,Z 466.046,A -85,B 0,C 180,E1 -25954.039,E2 -25954.039} C_VEL
LIN {X 0,Y 137.685,Z 473.324,A -85,B 0,C 180,E1 -25957.773,E2 -25957.773} C_VEL
LIN {X 0,Y 138.429,Z 478.031,A -85,B 0,C 180,E1 -25959.934,E2 -25959.934} C_VEL
LIN {X 0,Y 137.429,Z 486.495,A -85,B 0,C 180,E1 -25963.005,E2 -25963.005} C_VEL
LIN {X 0,Y 135.375,Z 495.888,A -85,B 0,C 180,E1 -25966.62,E2 -25966.62} C_VEL
LIN {X 0,Y 132.638,Z 504.768,A -85,B 0,C 180,E1 -25970.517,E2 -25970.517} C_VEL
LIN {X 0,Y 130.348,Z 509.383,A -85,B 0,C 180,E1 -25972.657,E2 -25972.657} C_VEL
LIN {X 0,Y 125.236,Z 517.217,A -85,B 0,C 180,E1 -25976.923,E2 -25976.923} C_VEL
LIN {X 0,Y 120.572,Z 524.257,A -85,B 0,C 180,E1 -25982.204,E2 -25982.204} C_VEL
LIN {X 0,Y 117.203,Z 529.018,A -85,B 0,C 180,E1 -25987.059,E2 -25987.059} C_VEL
LIN {X 0,Y 114.701,Z 532.669,A -85,B 0,C 180,E1 -25992.159,E2 -25992.159} C_VEL
LIN {X 0,Y 113.633,Z 534.566,A -85,B 0,C 180,E1 -25995.676,E2 -25995.676} C_VEL
LIN {X 0,Y 112.574,Z 537.027,A -85,B 0,C 180,E1 -26002.827,E2 -26002.827} C_VEL
LIN {X 0,Y 112.551,Z 537.779,A -85,B 0,C 180,E1 -26007.555,E2 -26007.555} C_VEL
LIN {X 0,Y 112.712,Z 537.896,A -85,B 0,C 180,E1 -26010,E2 -26010} C_VEL
LIN {X 0,Y 112.516,Z 537.649,A -85,B 0,C 180,E1 -26013.581,E2 -26013.581} C_VEL
LIN {X 0,Y 112.571,Z 537.004,A -85,B 0,C 180,E1 -26017.173,E2 -26017.173} C_VEL
LIN {X 0,Y 112.904,Z 535.965,A -85,B 0,C 180,E1 -26020.762,E2 -26020.762} C_VEL
LIN {X 0,Y 113.623,Z 534.521,A -85,B 0,C 180,E1 -26024.324,E2 -26024.324} C_VEL
LIN {X 0,Y 115.416,Z 531.515,A -85,B 0,C 180,E1 -26029.567,E2 -26029.567} C_VEL
LIN {X 0,Y 118.224,Z 527.479,A -85,B 0,C 180,E1 -26034.59,E2 -26034.59} C_VEL
LIN {X 0,Y 122.473,Z 521.289,A -85,B 0,C 180,E1 -26040.139,E2 -26040.139} C_VEL
LIN {X 0,Y 126.884,Z 514.543,A -85,B 0,C 180,E1 -26044.592,E2 -26044.592} C_VEL
LIN {X 0,Y 131.201,Z 507.699,A -85,B 0,C 180,E1 -26048.026,E2 -26048.026} C_VEL
LIN {X 0,Y 133.151,Z 502.888,A -85,B 0,C 180,E1 -26050.284,E2 -26050.284} C_VEL
LIN {X 0,Y 135.616,Z 494.526,A -85,B 0,C 180,E1 -26053.848,E2 -26053.848} C_VEL
LIN {X 0,Y 137.568,Z 484.978,A -85,B 0,C 180,E1 -26057.468,E2 -26057.468} C_VEL
LIN {X 0,Y 138.356,Z 477.75,A -85,B 0,C 180,E1 -26060.062,E2 -26060.062} C_VEL
LIN {X 0,Y 137.159,Z 471.563,A -85,B 0,C 180,E1 -26062.982,E2 -26062.982} C_VEL
LIN {X 0,Y 135.122,Z 464.408,A -85,B 0,C 180,E1 -26066.72,E2 -26066.72} C_VEL
LIN {X 0,Y 132.759,Z 457.64,A -85,B 0,C 180,E1 -26070.681,E2 -26070.681} C_VEL
LIN {X 0,Y 130.436,Z 452.115,A -85,B 0,C 180,E1 -26074.466,E2 -26074.466} C_VEL
LIN {X 0,Y 128.704,Z 448.076,A -85,B 0,C 180,E1 -26077.528,E2 -26077.528} C_VEL
LIN {X 0,Y 125.591,Z 441.856,A -85,B 0,C 180,E1 -26083.752,E2 -26083.752} C_VEL
LIN {X 0,Y 125.184,Z 440.598,A -85,B 0,C 180,E1 -26084.951,E2 -26084.951} C_VEL
LIN {X 0,Y 122.187,Z 435.579,A -85,B 0,C 180,E1 -26095.464,E2 -26095.464} C_VEL
LIN {X 0,Y 122.037,Z 434.004,A -85,B 0,C 180,E1 -26100,E2 -26100} C_VEL
LIN {X 0,Y 122.007,Z 435.002,A -85,B 0,C 180,E1 -26104.328,E2 -26104.328} C_VEL
LIN {X 0,Y 122.152,Z 436.405,A -85,B 0,C 180,E1 -26107.03,E2 -26107.03} C_VEL
LIN {X 0,Y 122.225,Z 440.615,A -85,B 0,C 180,E1 -26111.26,E2 -26111.26} C_VEL
LIN {X 0,Y 122.785,Z 446.069,A -85,B 0,C 180,E1 -26116.299,E2 -26116.299} C_VEL
LIN {X 0,Y 123.335,Z 447.37,A -85,B 0,C 180,E1 -26118.048,E2 -26118.048} C_VEL
LIN {X 0,Y 124.903,Z 449.525,A -85,B 0,C 180,E1 -26121.453,E2 -26121.453} C_VEL
LIN {X 0,Y 127.183,Z 453.944,A -85,B 0,C 180,E1 -26126.236,E2 -26126.236} C_VEL
LIN {X 0,Y 129.242,Z 458.354,A -85,B 0,C 180,E1 -26130.199,E2 -26130.199} C_VEL
LIN {X 0,Y 131.485,Z 463.977,A -85,B 0,C 180,E1 -26134.508,E2 -26134.508} C_VEL
LIN {X 0,Y 133.624,Z 470.814,A -85,B 0,C 180,E1 -26139.135,E2 -26139.135} C_VEL
LIN {X 0,Y 134.352,Z 475.703,A -85,B 0,C 180,E1 -26141.961,E2 -26141.961} C_VEL
LIN {X 0,Y 134.308,Z 482.2,A -85,B 0,C 180,E1 -26145.366,E2 -26145.366} C_VEL
LIN {X 0,Y 133.908,Z 485.919,A -85,B 0,C 180,E1 -26147.289,E2 -26147.289} C_VEL
LIN {X 0,Y 129.488,Z 493.774,A -85,B 0,C 180,E1 -26150.377,E2 -26150.377} C_VEL
LIN {X 0,Y 123.912,Z 501.981,A -85,B 0,C 180,E1 -26154.454,E2 -26154.454} C_VEL
LIN {X 0,Y 119.843,Z 507.583,A -85,B 0,C 180,E1 -26158.144,E2 -26158.144} C_VEL
LIN {X 0,Y 115.493,Z 513.044,A -85,B 0,C 180,E1 -26162.846,E2 -26162.846} C_VEL
LIN {X 0,Y 111.953,Z 517.32,A -85,B 0,C 180,E1 -26167.873,E2 -26167.873} C_VEL
LIN {X 0,Y 110.041,Z 519.58,A -85,B 0,C 180,E1 -26171.377,E2 -26171.377} C_VEL
LIN {X 0,Y 108.554,Z 521.409,A -85,B 0,C 180,E1 -26174.991,E2 -26174.991} C_VEL
LIN {X 0,Y 107.209,Z 523.028,A -85,B 0,C 180,E1 -26179.52,E2 -26179.52} C_VEL
LIN {X 0,Y 106.071,Z 524.358,A -85,B 0,C 180,E1 -26186.201,E2 -26186.201} C_VEL
LIN {X 0,Y 105.907,Z 524.581,A -85,B 0,C 180,E1 -26190,E2 -26190} C_VEL
LIN {X 0,Y 106.067,Z 524.385,A -85,B 0,C 180,E1 -26193.8,E2 -26193.8} C_VEL
LIN {X 0,Y 107.361,Z 522.844,A -85,B 0,C 180,E1 -26201.326,E2 -26201.326} C_VEL
LIN {X 0,Y 108.507,Z 521.499,A -85,B 0,C 180,E1 -26205.016,E2 -26205.016} C_VEL
LIN {X 0,Y 110.892,Z 518.654,A -85,B 0,C 180,E1 -26210.401,E2 -26210.401} C_VEL
LIN {X 0,Y 114.19,Z 514.781,A -85,B 0,C 180,E1 -26215.521,E2 -26215.521} C_VEL
LIN {X 0,Y 118.243,Z 509.782,A -85,B 0,C 180,E1 -26220.346,E2 -26220.346} C_VEL
LIN {X 0,Y 122.943,Z 503.482,A -85,B 0,C 180,E1 -26224.866,E2 -26224.866} C_VEL
LIN {X 0,Y 128.453,Z 495.582,A -85,B 0,C 180,E1 -26228.991,E2 -26228.991} C_VEL
LIN {X 0,Y 133.004,Z 488.054,A -85,B 0,C 180,E1 -26232.056,E2 -26232.056} C_VEL
LIN {X 0,Y 134.047,Z 485.788,A -85,B 0,C 180,E1 -26232.968,E2 -26232.968} C_VEL
LIN {X 0,Y 134.578,Z 479.474,A -85,B 0,C 180,E1 -26236.217,E2 -26236.217} C_VEL
LIN {X 0,Y 134.362,Z 474.734,A -85,B 0,C 180,E1 -26238.784,E2 -26238.784} C_VEL
LIN {X 0,Y 133.37,Z 469.885,A -85,B 0,C 180,E1 -26241.744,E2 -26241.744} C_VEL
LIN {X 0,Y 131.252,Z 463.32,A -85,B 0,C 180,E1 -26246.253,E2 -26246.253} C_VEL
LIN {X 0,Y 129.032,Z 457.654,A -85,B 0,C 180,E1 -26250.646,E2 -26250.646} C_VEL
LIN {X 0,Y 126.533,Z 452.812,A -85,B 0,C 180,E1 -26255.382,E2 -26255.382} C_VEL
LIN {X 0,Y 124.378,Z 448.675,A -85,B 0,C 180,E1 -26260.182,E2 -26260.182} C_VEL
LIN {X 0,Y 123.067,Z 446.7,A -85,B 0,C 180,E1 -26263.409,E2 -26263.409} C_VEL
LIN {X 0,Y 122.65,Z 445.327,A -85,B 0,C 180,E1 -26265.057,E2 -26265.057} C_VEL
LIN {X 0,Y 122.177,Z 444.364,A -85,B 0,C 180,E1 -26266.697,E2 -26266.697} C_VEL
LIN {X 0,Y 120.387,Z 441.4,A -85,B 0,C 180,E1 -26280,E2 -26280} C_VEL
LIN {X 0,Y 120.774,Z 443.727,A -85,B 0,C 180,E1 -26286.683,E2 -26286.683} C_VEL
LIN {X 0,Y 122.505,Z 446.72,A -85,B 0,C 180,E1 -26293.266,E2 -26293.266} C_VEL
LIN {X 0,Y 125.173,Z 453.088,A -85,B 0,C 180,E1 -26300.438,E2 -26300.438} C_VEL
LIN {X 0,Y 127.363,Z 459.018,A -85,B 0,C 180,E1 -26305.318,E2 -26305.318} C_VEL
LIN {X 0,Y 129.368,Z 465.325,A -85,B 0,C 180,E1 -26309.632,E2 -26309.632} C_VEL
LIN {X 0,Y 131.106,Z 471.332,A -85,B 0,C 180,E1 -26313.34,E2 -26313.34} C_VEL
LIN {X 0,Y 132.423,Z 477.305,A -85,B 0,C 180,E1 -26316.66,E2 -26316.66} C_VEL
LIN {X 0,Y 132.809,Z 481.869,A -85,B 0,C 180,E1 -26318.883,E2 -26318.883} C_VEL
LIN {X 0,Y 131.069,Z 491.086,A -85,B 0,C 180,E1 -26322.5,E2 -26322.5} C_VEL
LIN {X 0,Y 128.769,Z 499.098,A -85,B 0,C 180,E1 -26325.902,E2 -26325.902} C_VEL
LIN {X 0,Y 126.325,Z 505.93,A -85,B 0,C 180,E1 -26329.178,E2 -26329.178} C_VEL
LIN {X 0,Y 123.798,Z 510.331,A -85,B 0,C 180,E1 -26331.356,E2 -26331.356} C_VEL
LIN {X 0,Y 118.418,Z 518.026,A -85,B 0,C 180,E1 -26335.885,E2 -26335.885} C_VEL
LIN {X 0,Y 114.312,Z 523.824,A -85,B 0,C 180,E1 -26340.537,E2 -26340.537} C_VEL
LIN {X 0,Y 110.658,Z 528.584,A -85,B 0,C 180,E1 -26345.617,E2 -26345.617} C_VEL
LIN {X 0,Y 107.916,Z 532.235,A -85,B 0,C 180,E1 -26350.996,E2 -26350.996} C_VEL
LIN {X 0,Y 106.727,Z 534.132,A -85,B 0,C 180,E1 -26354.728,E2 -26354.728} C_VEL
LIN {X 0,Y 105.507,Z 536.593,A -85,B 0,C 180,E1 -26362.344,E2 -26362.344} C_VEL
LIN {X 0,Y 105.491,Z 537.373,A -85,B 0,C 180,E1 -26367.896,E2 -26367.896} C_VEL
LIN {X 0,Y 105.615,Z 537.464,A -85,B 0,C 180,E1 -26370,E2 -26370} C_VEL
LIN {X 0,Y 105.417,Z 537.216,A -85,B 0,C 180,E1 -26373.822,E2 -26373.822} C_VEL
LIN {X 0,Y 105.505,Z 536.57,A -85,B 0,C 180,E1 -26377.656,E2 -26377.656} C_VEL
LIN {X 0,Y 106.719,Z 534.085,A -85,B 0,C 180,E1 -26385.273,E2 -26385.273} C_VEL
LIN {X 0,Y 108.729,Z 531.08,A -85,B 0,C 180,E1 -26390.824,E2 -26390.824} C_VEL
LIN {X 0,Y 111.752,Z 527.042,A -85,B 0,C 180,E1 -26396.118,E2 -26396.118} C_VEL
LIN {X 0,Y 115.658,Z 521.866,A -85,B 0,C 180,E1 -26401.098,E2 -26401.098} C_VEL
LIN {X 0,Y 121.079,Z 514.106,A -85,B 0,C 180,E1 -26406.51,E2 -26406.51} C_VEL
LIN {X 0,Y 125.555,Z 507.253,A -85,B 0,C 180,E1 -26410.069,E2 -26410.069} C_VEL
LIN {X 0,Y 128.604,Z 499.349,A -85,B 0,C 180,E1 -26413.881,E2 -26413.881} C_VEL
LIN {X 0,Y 131.26,Z 489.69,A -85,B 0,C 180,E1 -26417.979,E2 -26417.979} C_VEL
LIN {X 0,Y 132.744,Z 481.569,A -85,B 0,C 180,E1 -26421.126,E2 -26421.126} C_VEL
LIN {X 0,Y 132.805,Z 480.191,A -85,B 0,C 180,E1 -26421.713,E2 -26421.713} C_VEL
LIN {X 0,Y 131.272,Z 472.249,A -85,B 0,C 180,E1 -26425.992,E2 -26425.992} C_VEL
LIN {X 0,Y 129.417,Z 465.755,A -85,B 0,C 180,E1 -26429.937,E2 -26429.937} C_VEL
LIN {X 0,Y 128.327,Z 462.256,A -85,B 0,C 180,E1 -26432.257,E2 -26432.257} C_VEL
LIN {X 0,Y 126.818,Z 457.819,A -85,B 0,C 180,E1 -26435.441,E2 -26435.441} C_VEL
LIN {X 0,Y 125.248,Z 453.569,A -85,B 0,C 180,E1 -26438.916,E2 -26438.916} C_VEL
LIN {X 0,Y 123.28,Z 449.466,A -85,B 0,C 180,E1 -26443.439,E2 -26443.439} C_VEL
LIN {X 0,Y 122.825,Z 447.715,A -85,B 0,C 180,E1 -26445.079,E2 -26445.079} C_VEL
LIN {X 0,Y 122.265,Z 446.592,A -85,B 0,C 180,E1 -26446.707,E2 -26446.707} C_VEL
LIN {X 0,Y 120.209,Z 442.087,A -85,B 0,C 180,E1 -26456.648,E2 -26456.648} C_VEL
LIN {X 0,Y 120.207,Z 440.94,A -85,B 0,C 180,E1 -26460,E2 -26460} C_VEL
LIN {X 0,Y 121.904,Z 444.197,A -85,B 0,C 180,E1 -26473.333,E2 -26473.333} C_VEL
LIN {X 0,Y 122.462,Z 444.898,A -85,B 0,C 180,E1 -26474.967,E2 -26474.967} C_VEL
LIN {X 0,Y 123.335,Z 447.37,A -85,B 0,C 180,E1 -26478.048,E2 -26478.048} C_VEL
LIN {X 0,Y 124.161,Z 449.636,A -85,B 0,C 180,E1 -26480.541,E2 -26480.541} C_VEL
LIN {X 0,Y 124.563,Z 452.865,A -85,B 0,C 180,E1 -26482.833,E2 -26482.833} C_VEL
LIN {X 0,Y 124.905,Z 462.724,A -85,B 0,C 180,E1 -26488.706,E2 -26488.706} C_VEL
LIN {X 0,Y 125.382,Z 464.795,A -85,B 0,C 180,E1 -26490.278,E2 -26490.278} C_VEL
LIN {X 0,Y 127.388,Z 471.18,A -85,B 0,C 180,E1 -26495.399,E2 -26495.399} C_VEL
LIN {X 0,Y 128.576,Z 476.318,A -85,B 0,C 180,E1 -26499.051,E2 -26499.051} C_VEL
LIN {X 0,Y 128.725,Z 482.3,A -85,B 0,C 180,E1 -26502.613,E2 -26502.613} C_VEL
LIN {X 0,Y 128.067,Z 487.455,A -85,B 0,C 180,E1 -26505.513,E2 -26505.513} C_VEL
LIN {X 0,Y 125.108,Z 492.626,A -85,B 0,C 180,E1 -26507.616,E2 -26507.616} C_VEL
LIN {X 0,Y 119.133,Z 501.196,A -85,B 0,C 180,E1 -26511.726,E2 -26511.726} C_VEL
LIN {X 0,Y 113.882,Z 508.016,A -85,B 0,C 180,E1 -26516.261,E2 -26516.261} C_VEL
LIN {X 0,Y 109.239,Z 513.477,A -85,B 0,C 180,E1 -26521.15,E2 -26521.15} C_VEL
LIN {X 0,Y 105.411,Z 517.754,A -85,B 0,C 180,E1 -26526.42,E2 -26526.42} C_VEL
LIN {X 0,Y 103.352,Z 520.012,A -85,B 0,C 180,E1 -26530.123,E2 -26530.123} C_VEL
LIN {X 0,Y 101.735,Z 521.841,A -85,B 0,C 180,E1 -26533.959,E2 -26533.959} C_VEL
LIN {X 0,Y 100.091,Z 523.638,A -85,B 0,C 180,E1 -26539.429,E2 -26539.429} C_VEL
LIN {X 0,Y 99.017,Z 524.789,A -85,B 0,C 180,E1 -26545.93,E2 -26545.93} C_VEL
LIN {X 0,Y 98.836,Z 525.012,A -85,B 0,C 180,E1 -26550,E2 -26550} C_VEL
LIN {X 0,Y 99.012,Z 524.815,A -85,B 0,C 180,E1 -26554.071,E2 -26554.071} C_VEL
LIN {X 0,Y 100.425,Z 523.275,A -85,B 0,C 180,E1 -26562.12,E2 -26562.12} C_VEL
LIN {X 0,Y 101.677,Z 521.93,A -85,B 0,C 180,E1 -26566.051,E2 -26566.051} C_VEL
LIN {X 0,Y 104.29,Z 519.083,A -85,B 0,C 180,E1 -26571.756,E2 -26571.756} C_VEL
LIN {X 0,Y 107.827,Z 515.213,A -85,B 0,C 180,E1 -26577.146,E2 -26577.146} C_VEL
LIN {X 0,Y 112.191,Z 510.212,A -85,B 0,C 180,E1 -26582.173,E2 -26582.173} C_VEL
LIN {X 0,Y 117.203,Z 503.911,A -85,B 0,C 180,E1 -26586.845,E2 -26586.845} C_VEL
LIN {X 0,Y 123.027,Z 496.011,A -85,B 0,C 180,E1 -26591.068,E2 -26591.068} C_VEL
LIN {X 0,Y 127.235,Z 489.508,A -85,B 0,C 180,E1 -26593.805,E2 -26593.805} C_VEL
LIN {X 0,Y 128.129,Z 487.754,A -85,B 0,C 180,E1 -26594.515,E2 -26594.515} C_VEL
LIN {X 0,Y 128.896,Z 481.134,A -85,B 0,C 180,E1 -26598.246,E2 -26598.246} C_VEL
LIN {X 0,Y 128.699,Z 476.876,A -85,B 0,C 180,E1 -26600.844,E2 -26600.844} C_VEL
LIN {X 0,Y 127.51,Z 471.502,A -85,B 0,C 180,E1 -26604.64,E2 -26604.64} C_VEL
LIN {X 0,Y 125.543,Z 465.129,A -85,B 0,C 180,E1 -26609.746,E2 -26609.746} C_VEL
LIN {X 0,Y 124.119,Z 461.591,A -85,B 0,C 180,E1 -26613.064,E2 -26613.064} C_VEL
LIN {X 0,Y 122.767,Z 458.469,A -85,B 0,C 180,E1 -26616.376,E2 -26616.376} C_VEL
LIN {X 0,Y 121.605,Z 455.643,A -85,B 0,C 180,E1 -26619.71,E2 -26619.71} C_VEL
LIN {X 0,Y 119.672,Z 451.285,A -85,B 0,C 180,E1 -26626.414,E2 -26626.414} C_VEL
LIN {X 0,Y 118.003,Z 448.768,A -85,B 0,C 180,E1 -26636.585,E2 -26636.585} C_VEL
LIN {X 0,Y 118.169,Z 448.191,A -85,B 0,C 180,E1 -26640,E2 -26640} C_VEL
LIN {X 0,Y 118.413,Z 450.589,A -85,B 0,C 180,E1 -26646.817,E2 -26646.817} C_VEL
LIN {X 0,Y 119.958,Z 453.892,A -85,B 0,C 180,E1 -26653.553,E2 -26653.553} C_VEL
LIN {X 0,Y 121.936,Z 459.9,A -85,B 0,C 180,E1 -26660.232,E2 -26660.232} C_VEL
LIN {X 0,Y 123.403,Z 464.536,A -85,B 0,C 180,E1 -26664.323,E2 -26664.323} C_VEL
LIN {X 0,Y 125.295,Z 471.777,A -85,B 0,C 180,E1 -26669.601,E2 -26669.601} C_VEL
LIN {X 0,Y 126.861,Z 479.655,A -85,B 0,C 180,E1 -26674.6,E2 -26674.6} C_VEL
LIN {X 0,Y 127.236,Z 484.762,A -85,B 0,C 180,E1 -26677.416,E2 -26677.416} C_VEL
LIN {X 0,Y 125.006,Z 493.788,A -85,B 0,C 180,E1 -26681.239,E2 -26681.239} C_VEL
LIN {X 0,Y 122.607,Z 500.859,A -85,B 0,C 180,E1 -26684.485,E2 -26684.485} C_VEL
LIN {X 0,Y 120.084,Z 507.004,A -85,B 0,C 180,E1 -26687.696,E2 -26687.696} C_VEL
LIN {X 0,Y 116.366,Z 512.587,A -85,B 0,C 180,E1 -26690.642,E2 -26690.642} C_VEL
LIN {X 0,Y 110.965,Z 519.682,A -85,B 0,C 180,E1 -26695.422,E2 -26695.422} C_VEL
LIN {X 0,Y 106.705,Z 525.096,A -85,B 0,C 180,E1 -26700.397,E2 -26700.397} C_VEL
LIN {X 0,Y 103.108,Z 529.476,A -85,B 0,C 180,E1 -26705.859,E2 -26705.859} C_VEL
LIN {X 0,Y 101.188,Z 531.8,A -85,B 0,C 180,E1 -26709.679,E2 -26709.679} C_VEL
LIN {X 0,Y 99.84,Z 533.697,A -85,B 0,C 180,E1 -26713.645,E2 -26713.645} C_VEL
LIN {X 0,Y 98.451,Z 536.16,A -85,B 0,C 180,E1 -26721.791,E2 -26721.791} C_VEL
LIN {X 0,Y 98.43,Z 536.971,A -85,B 0,C 180,E1 -26728.416,E2 -26728.416} C_VEL
LIN {X 0,Y 98.432,Z 536.964,A -85,B 0,C 180,E1 -26731.634,E2 -26731.634} C_VEL
LIN {X 0,Y 98.449,Z 536.136,A -85,B 0,C 180,E1 -26738.208,E2 -26738.208} C_VEL
LIN {X 0,Y 98.922,Z 535.095,A -85,B 0,C 180,E1 -26742.306,E2 -26742.306} C_VEL
LIN {X 0,Y 99.833,Z 533.649,A -85,B 0,C 180,E1 -26746.355,E2 -26746.355} C_VEL
LIN {X 0,Y 102.081,Z 530.644,A -85,B 0,C 180,E1 -26752.251,E2 -26752.251} C_VEL
LIN {X 0,Y 105.376,Z 526.605,A -85,B 0,C 180,E1 -26757.831,E2 -26757.831} C_VEL
LIN {X 0,Y 109.448,Z 521.585,A -85,B 0,C 180,E1 -26762.897,E2 -26762.897} C_VEL
LIN {X 0,Y 114.495,Z 514.913,A -85,B 0,C 180,E1 -26767.867,E2 -26767.867} C_VEL
LIN {X 0,Y 119.235,Z 508.32,A -85,B 0,C 180,E1 -26771.537,E2 -26771.537} C_VEL
LIN {X 0,Y 122.584,Z 500.715,A -85,B 0,C 180,E1 -26775.469,E2 -26775.469} C_VEL
LIN {X 0,Y 125.563,Z 491.418,A -85,B 0,C 180,E1 -26779.695,E2 -26779.695} C_VEL
LIN {X 0,Y 127.164,Z 484.559,A -85,B 0,C 180,E1 -26782.559,E2 -26782.559} C_VEL
LIN {X 0,Y 126.747,Z 479.494,A -85,B 0,C 180,E1 -26785.365,E2 -26785.365} C_VEL
LIN {X 0,Y 125.427,Z 472.535,A -85,B 0,C 180,E1 -26789.716,E2 -26789.716} C_VEL
LIN {X 0,Y 123.798,Z 466.61,A -85,B 0,C 180,E1 -26793.989,E2 -26793.989} C_VEL
LIN {X 0,Y 122.983,Z 463.368,A -85,B 0,C 180,E1 -26796.42,E2 -26796.42} C_VEL
LIN {X 0,Y 121.807,Z 459.589,A -85,B 0,C 180,E1 -26799.746,E2 -26799.746} C_VEL
LIN {X 0,Y 119.787,Z 453.602,A -85,B 0,C 180,E1 -26806.427,E2 -26806.427} C_VEL
LIN {X 0,Y 118.229,Z 450.293,A -85,B 0,C 180,E1 -26813.172,E2 -26813.172} C_VEL
LIN {X 0,Y 118.007,Z 447.755,A -85,B 0,C 180,E1 -26820,E2 -26820} C_VEL
LIN {X 0,Y 119.46,Z 450.984,A -85,B 0,C 180,E1 -26833.611,E2 -26833.611} C_VEL
LIN {X 0,Y 120.293,Z 453.663,A -85,B 0,C 180,E1 -26837.452,E2 -26837.452} C_VEL
LIN {X 0,Y 121.397,Z 455.363,A -85,B 0,C 180,E1 -26840.326,E2 -26840.326} C_VEL
LIN {X 0,Y 123.308,Z 459.571,A -85,B 0,C 180,E1 -26845.307,E2 -26845.307} C_VEL
LIN {X 0,Y 125.382,Z 464.795,A -85,B 0,C 180,E1 -26850.278,E2 -26850.278} C_VEL
LIN {X 0,Y 125.967,Z 468.01,A -85,B 0,C 180,E1 -26852.533,E2 -26852.533} C_VEL
LIN {X 0,Y 125.612,Z 473.185,A -85,B 0,C 180,E1 -26855.276,E2 -26855.276} C_VEL
LIN {X 0,Y 124.048,Z 480.209,A -85,B 0,C 180,E1 -26858.586,E2 -26858.586} C_VEL
LIN {X 0,Y 122.939,Z 485.479,A -85,B 0,C 180,E1 -26861.415,E2 -26861.415} C_VEL
LIN {X 0,Y 122.321,Z 489.044,A -85,B 0,C 180,E1 -26863.588,E2 -26863.588} C_VEL
LIN {X 0,Y 120.745,Z 491.906,A -85,B 0,C 180,E1 -26864.857,E2 -26864.857} C_VEL
LIN {X 0,Y 114.708,Z 500.307,A -85,B 0,C 180,E1 -26868.804,E2 -26868.804} C_VEL
LIN {X 0,Y 108.963,Z 507.431,A -85,B 0,C 180,E1 -26873.372,E2 -26873.372} C_VEL
LIN {X 0,Y 104.67,Z 512.231,A -85,B 0,C 180,E1 -26877.51,E2 -26877.51} C_VEL
LIN {X 0,Y 100.242,Z 516.889,A -85,B 0,C 180,E1 -26882.889,E2 -26882.889} C_VEL
LIN {X 0,Y 96.73,Z 520.444,A -85,B 0,C 180,E1 -26888.699,E2 -26888.699} C_VEL
LIN {X 0,Y 94.943,Z 522.274,A -85,B 0,C 180,E1 -26892.777,E2 -26892.777} C_VEL
LIN {X 0,Y 93.038,Z 524.194,A -85,B 0,C 180,E1 -26899.117,E2 -26899.117} C_VEL
LIN {X 0,Y 91.967,Z 525.22,A -85,B 0,C 180,E1 -26905.618,E2 -26905.618} C_VEL
LIN {X 0,Y 91.766,Z 525.443,A -85,B 0,C 180,E1 -26910,E2 -26910} C_VEL
LIN {X 0,Y 91.961,Z 525.246,A -85,B 0,C 180,E1 -26914.384,E2 -26914.384} C_VEL
LIN {X 0,Y 93.513,Z 523.706,A -85,B 0,C 180,E1 -26923.031,E2 -26923.031} C_VEL
LIN {X 0,Y 94.874,Z 522.361,A -85,B 0,C 180,E1 -26927.237,E2 -26927.237} C_VEL
LIN {X 0,Y 97.735,Z 519.515,A -85,B 0,C 180,E1 -26933.298,E2 -26933.298} C_VEL
LIN {X 0,Y 101.57,Z 515.643,A -85,B 0,C 180,E1 -26938.971,E2 -26938.971} C_VEL
LIN {X 0,Y 106.266,Z 510.642,A -85,B 0,C 180,E1 -26944.206,E2 -26944.206} C_VEL
LIN {X 0,Y 111.62,Z 504.34,A -85,B 0,C 180,E1 -26949.024,E2 -26949.024} C_VEL
LIN {X 0,Y 117.781,Z 496.439,A -85,B 0,C 180,E1 -26953.331,E2 -26953.331} C_VEL
LIN {X 0,Y 121.561,Z 490.984,A -85,B 0,C 180,E1 -26955.688,E2 -26955.688} C_VEL
LIN {X 0,Y 122.42,Z 489.289,A -85,B 0,C 180,E1 -26956.456,E2 -26956.456} C_VEL
LIN {X 0,Y 123.176,Z 484.511,A -85,B 0,C 180,E1 -26959.387,E2 -26959.387} C_VEL
LIN {X 0,Y 123.16,Z 480.41,A -85,B 0,C 180,E1 -26962.16,E2 -26962.16} C_VEL
LIN {X 0,Y 122.338,Z 475.566,A -85,B 0,C 180,E1 -26965.942,E2 -26965.942} C_VEL
LIN {X 0,Y 120.998,Z 470.258,A -85,B 0,C 180,E1 -26970.606,E2 -26970.606} C_VEL
LIN {X 0,Y 119.4,Z 465.363,A -85,B 0,C 180,E1 -26975.667,E2 -26975.667} C_VEL
LIN {X 0,Y 117.896,Z 461.309,A -85,B 0,C 180,E1 -26980.861,E2 -26980.861} C_VEL
LIN {X 0,Y 116.673,Z 458.217,A -85,B 0,C 180,E1 -26986.057,E2 -26986.057} C_VEL
LIN {X 0,Y 115.994,Z 456.903,A -85,B 0,C 180,E1 -26989.527,E2 -26989.527} C_VEL
LIN {X 0,Y 115.528,Z 454.85,A -85,B 0,C 180,E1 -27000,E2 -27000} C_VEL
LIN {X 0,Y 115.673,Z 457.304,A -85,B 0,C 180,E1 -27006.979,E2 -27006.979} C_VEL
LIN {X 0,Y 116.642,Z 459.736,A -85,B 0,C 180,E1 -27012.174,E2 -27012.174} C_VEL
LIN {X 0,Y 118.145,Z 465.426,A -85,B 0,C 180,E1 -27019.097,E2 -27019.097} C_VEL
LIN {X 0,Y 119.27,Z 470.03,A -85,B 0,C 180,E1 -27023.437,E2 -27023.437} C_VEL
LIN {X 0,Y 120.733,Z 477.383,A -85,B 0,C 180,E1 -27029.17,E2 -27029.17} C_VEL
LIN {X 0,Y 121.61,Z 484.286,A -85,B 0,C 180,E1 -27033.863,E2 -27033.863} C_VEL
LIN {X 0,Y 121.584,Z 487.911,A -85,B 0,C 180,E1 -27035.976,E2 -27035.976} C_VEL
LIN {X 0,Y 119,Z 496.328,A -85,B 0,C 180,E1 -27039.846,E2 -27039.846} C_VEL
LIN {X 0,Y 115.415,Z 505.024,A -85,B 0,C 180,E1 -27044.315,E2 -27044.315} C_VEL
LIN {X 0,Y 112.976,Z 509.464,A -85,B 0,C 180,E1 -27046.819,E2 -27046.819} C_VEL
LIN {X 0,Y 107.07,Z 516.933,A -85,B 0,C 180,E1 -27051.422,E2 -27051.422} C_VEL
LIN {X 0,Y 102.095,Z 522.956,A -85,B 0,C 180,E1 -27056.584,E2 -27056.584} C_VEL
LIN {X 0,Y 97.827,Z 527.717,A -85,B 0,C 180,E1 -27062.162,E2 -27062.162} C_VEL
LIN {X 0,Y 94.52,Z 531.366,A -85,B 0,C 180,E1 -27068.174,E2 -27068.174} C_VEL
LIN {X 0,Y 93.004,Z 533.262,A -85,B 0,C 180,E1 -27072.406,E2 -27072.406} C_VEL
LIN {X 0,Y 91.986,Z 534.695,A -85,B 0,C 180,E1 -27076.749,E2 -27076.749} C_VEL
LIN {X 0,Y 91.394,Z 535.726,A -85,B 0,C 180,E1 -27081.153,E2 -27081.153} C_VEL
LIN {X 0,Y 91.378,Z 536.569,A -85,B 0,C 180,E1 -27089.009,E2 -27089.009} C_VEL
LIN {X 0,Y 91.23,Z 536.349,A -85,B 0,C 180,E1 -27094.418,E2 -27094.418} C_VEL
LIN {X 0,Y 91.391,Z 535.701,A -85,B 0,C 180,E1 -27098.847,E2 -27098.847} C_VEL
LIN {X 0,Y 91.952,Z 534.659,A -85,B 0,C 180,E1 -27103.255,E2 -27103.255} C_VEL
LIN {X 0,Y 92.998,Z 533.213,A -85,B 0,C 180,E1 -27107.595,E2 -27107.595} C_VEL
LIN {X 0,Y 95.512,Z 530.208,A -85,B 0,C 180,E1 -27113.872,E2 -27113.872} C_VEL
LIN {X 0,Y 99.111,Z 526.169,A -85,B 0,C 180,E1 -27119.76,E2 -27119.76} C_VEL
LIN {X 0,Y 103.848,Z 520.685,A -85,B 0,C 180,E1 -27125.477,E2 -27125.477} C_VEL
LIN {X 0,Y 109.927,Z 513.232,A -85,B 0,C 180,E1 -27130.944,E2 -27130.944} C_VEL
LIN {X 0,Y 113.857,Z 507.871,A -85,B 0,C 180,E1 -27133.981,E2 -27133.981} C_VEL
LIN {X 0,Y 117.102,Z 500.834,A -85,B 0,C 180,E1 -27137.831,E2 -27137.831} C_VEL
LIN {X 0,Y 120.299,Z 492.025,A -85,B 0,C 180,E1 -27142.063,E2 -27142.063} C_VEL
LIN {X 0,Y 121.553,Z 487.605,A -85,B 0,C 180,E1 -27144.043,E2 -27144.043} C_VEL
LIN {X 0,Y 121.478,Z 483.906,A -85,B 0,C 180,E1 -27146.248,E2 -27146.248} C_VEL
LIN {X 0,Y 120.568,Z 476.96,A -85,B 0,C 180,E1 -27150.969,E2 -27150.969} C_VEL
LIN {X 0,Y 119.183,Z 470.332,A -85,B 0,C 180,E1 -27156.166,E2 -27156.166} C_VEL
LIN {X 0,Y 118.923,Z 468.775,A -85,B 0,C 180,E1 -27157.41,E2 -27157.41} C_VEL
LIN {X 0,Y 118.022,Z 465.134,A -85,B 0,C 180,E1 -27160.882,E2 -27160.882} C_VEL
LIN {X 0,Y 116.477,Z 459.464,A -85,B 0,C 180,E1 -27167.808,E2 -27167.808} C_VEL
LIN {X 0,Y 115.278,Z 455.631,A -85,B 0,C 180,E1 -27176.505,E2 -27176.505} C_VEL
LIN {X 0,Y 115.397,Z 454.442,A -85,B 0,C 180,E1 -27180,E2 -27180} C_VEL
LIN {X 0,Y 115.785,Z 456.642,A -85,B 0,C 180,E1 -27190.492,E2 -27190.492} C_VEL
LIN {X 0,Y 116.514,Z 457.876,A -85,B 0,C 180,E1 -27193.962,E2 -27193.962} C_VEL
LIN {X 0,Y 118.148,Z 462.338,A -85,B 0,C 180,E1 -27200.911,E2 -27200.911} C_VEL
LIN {X 0,Y 119.239,Z 465.053,A -85,B 0,C 180,E1 -27204.367,E2 -27204.367} C_VEL
LIN {X 0,Y 121.143,Z 470.851,A -85,B 0,C 180,E1 -27210.3,E2 -27210.3} C_VEL
LIN {X 0,Y 122.467,Z 476.386,A -85,B 0,C 180,E1 -27215.021,E2 -27215.021} C_VEL
LIN {X 0,Y 123.095,Z 480.016,A -85,B 0,C 180,E1 -27217.835,E2 -27217.835} C_VEL
LIN {X 0,Y 122.973,Z 485.224,A -85,B 0,C 180,E1 -27221.263,E2 -27221.263} C_VEL
LIN {X 0,Y 122.939,Z 485.479,A -85,B 0,C 180,E1 -27221.415,E2 -27221.415} C_VEL
LIN {X 0,Y 122.321,Z 487.2,A -85,B 0,C 180,E1 -27222.249,E2 -27222.249} C_VEL
LIN {X 0,Y 120.34,Z 489.985,A -85,B 0,C 180,E1 -27223.149,E2 -27223.149} C_VEL
LIN {X 0,Y 111.756,Z 498.175,A -85,B 0,C 180,E1 -27225.119,E2 -27225.119} C_VEL
LIN {X 0,Y 110.17,Z 499.888,A -85,B 0,C 180,E1 -27225.901,E2 -27225.901} C_VEL
LIN {X 0,Y 104.281,Z 506.765,A -85,B 0,C 180,E1 -27230.19,E2 -27230.19} C_VEL
LIN {X 0,Y 98.772,Z 512.663,A -85,B 0,C 180,E1 -27235.304,E2 -27235.304} C_VEL
LIN {X 0,Y 93.995,Z 517.322,A -85,B 0,C 180,E1 -27240.922,E2 -27240.922} C_VEL
LIN {X 0,Y 90.161,Z 520.877,A -85,B 0,C 180,E1 -27247.062,E2 -27247.062} C_VEL
LIN {X 0,Y 88.187,Z 522.707,A -85,B 0,C 180,E1 -27251.411,E2 -27251.411} C_VEL
LIN {X 0,Y 85.893,Z 524.804,A -85,B 0,C 180,E1 -27259.076,E2 -27259.076} C_VEL
LIN {X 0,Y 84.901,Z 525.652,A -85,B 0,C 180,E1 -27265.252,E2 -27265.252} C_VEL
LIN {X 0,Y 84.698,Z 525.873,A -85,B 0,C 180,E1 -27270,E2 -27270} C_VEL
LIN {X 0,Y 84.894,Z 525.677,A -85,B 0,C 180,E1 -27274.749,E2 -27274.749} C_VEL
LIN {X 0,Y 86.615,Z 524.137,A -85,B 0,C 180,E1 -27284.089,E2 -27284.089} C_VEL
LIN {X 0,Y 88.137,Z 522.792,A -85,B 0,C 180,E1 -27288.601,E2 -27288.601} C_VEL
LIN {X 0,Y 91.271,Z 519.945,A -85,B 0,C 180,E1 -27295.057,E2 -27295.057} C_VEL
LIN {X 0,Y 95.436,Z 516.073,A -85,B 0,C 180,E1 -27301.031,E2 -27301.031} C_VEL
LIN {X 0,Y 100.491,Z 511.071,A -85,B 0,C 180,E1 -27306.475,E2 -27306.475} C_VEL
LIN {X 0,Y 106.218,Z 504.768,A -85,B 0,C 180,E1 -27311.428,E2 -27311.428} C_VEL
LIN {X 0,Y 112.738,Z 496.868,A -85,B 0,C 180,E1 -27315.8,E2 -27315.8} C_VEL
LIN {X 0,Y 115.938,Z 492.508,A -85,B 0,C 180,E1 -27317.729,E2 -27317.729} C_VEL
LIN {X 0,Y 116.811,Z 490.891,A -85,B 0,C 180,E1 -27318.561,E2 -27318.561} C_VEL
LIN {X 0,Y 117.628,Z 486.122,A -85,B 0,C 180,E1 -27321.817,E2 -27321.817} C_VEL
LIN {X 0,Y 117.419,Z 481.759,A -85,B 0,C 180,E1 -27325.348,E2 -27325.348} C_VEL
LIN {X 0,Y 116.68,Z 477.342,A -85,B 0,C 180,E1 -27329.404,E2 -27329.404} C_VEL
LIN {X 0,Y 115.975,Z 473.779,A -85,B 0,C 180,E1 -27332.967,E2 -27332.967} C_VEL
LIN {X 0,Y 114.643,Z 469.391,A -85,B 0,C 180,E1 -27338.419,E2 -27338.419} C_VEL
LIN {X 0,Y 113.968,Z 466.87,A -85,B 0,C 180,E1 -27342.041,E2 -27342.041} C_VEL
LIN {X 0,Y 113.293,Z 464.909,A -85,B 0,C 180,E1 -27345.633,E2 -27345.633} C_VEL
LIN {X 0,Y 112.813,Z 463.396,A -85,B 0,C 180,E1 -27349.228,E2 -27349.228} C_VEL
LIN {X 0,Y 112.458,Z 461.399,A -85,B 0,C 180,E1 -27359.286,E2 -27359.286} C_VEL
LIN {X 0,Y 112.456,Z 461.557,A -85,B 0,C 180,E1 -27360.623,E2 -27360.623} C_VEL
LIN {X 0,Y 112.561,Z 463.873,A -85,B 0,C 180,E1 -27367.173,E2 -27367.173} C_VEL
LIN {X 0,Y 113.089,Z 465.422,A -85,B 0,C 180,E1 -27370.745,E2 -27370.745} C_VEL
LIN {X 0,Y 114.133,Z 470.801,A -85,B 0,C 180,E1 -27377.932,E2 -27377.932} C_VEL
LIN {X 0,Y 114.894,Z 475.448,A -85,B 0,C 180,E1 -27382.593,E2 -27382.593} C_VEL
LIN {X 0,Y 115.771,Z 481.907,A -85,B 0,C 180,E1 -27388.065,E2 -27388.065} C_VEL
LIN {X 0,Y 116.178,Z 488.565,A -85,B 0,C 180,E1 -27392.986,E2 -27392.986} C_VEL
LIN {X 0,Y 116.132,Z 489.995,A -85,B 0,C 180,E1 -27393.933,E2 -27393.933} C_VEL
LIN {X 0,Y 114.174,Z 495.858,A -85,B 0,C 180,E1 -27396.848,E2 -27396.848} C_VEL
LIN {X 0,Y 111.04,Z 502.944,A -85,B 0,C 180,E1 -27400.578,E2 -27400.578} C_VEL
LIN {X 0,Y 107.816,Z 509.026,A -85,B 0,C 180,E1 -27404.188,E2 -27404.188} C_VEL
LIN {X 0,Y 101.585,Z 516.5,A -85,B 0,C 180,E1 -27408.909,E2 -27408.909} C_VEL
LIN {X 0,Y 96.176,Z 522.52,A -85,B 0,C 180,E1 -27414.225,E2 -27414.225} C_VEL
LIN {X 0,Y 91.577,Z 527.283,A -85,B 0,C 180,E1 -27420.076,E2 -27420.076} C_VEL
LIN {X 0,Y 87.929,Z 530.932,A -85,B 0,C 180,E1 -27426.444,E2 -27426.444} C_VEL
LIN {X 0,Y 86.228,Z 532.828,A -85,B 0,C 180,E1 -27430.972,E2 -27430.972} C_VEL
LIN {X 0,Y 84.37,Z 535.292,A -85,B 0,C 180,E1 -27440.409,E2 -27440.409} C_VEL
LIN {X 0,Y 84.34,Z 536.159,A -85,B 0,C 180,E1 -27449.463,E2 -27449.463} C_VEL
LIN {X 0,Y 84.151,Z 535.916,A -85,B 0,C 180,E1 -27454.79,E2 -27454.79} C_VEL
LIN {X 0,Y 84.364,Z 535.267,A -85,B 0,C 180,E1 -27459.59,E2 -27459.59} C_VEL
LIN {X 0,Y 86.223,Z 532.777,A -85,B 0,C 180,E1 -27469.028,E2 -27469.028} C_VEL
LIN {X 0,Y 89.034,Z 529.773,A -85,B 0,C 180,E1 -27475.731,E2 -27475.731} C_VEL
LIN {X 0,Y 92.979,Z 525.732,A -85,B 0,C 180,E1 -27481.945,E2 -27481.945} C_VEL
LIN {X 0,Y 98.392,Z 519.901,A -85,B 0,C 180,E1 -27488.213,E2 -27488.213} C_VEL
LIN {X 0,Y 104.648,Z 512.796,A -85,B 0,C 180,E1 -27493.501,E2 -27493.501} C_VEL
LIN {X 0,Y 107.788,Z 508.836,A -85,B 0,C 180,E1 -27495.825,E2 -27495.825} C_VEL
LIN {X 0,Y 111.563,Z 501.516,A -85,B 0,C 180,E1 -27500.101,E2 -27500.101} C_VEL
LIN {X 0,Y 114.699,Z 493.999,A -85,B 0,C 180,E1 -27503.96,E2 -27503.96} C_VEL
LIN {X 0,Y 116.081,Z 489.685,A -85,B 0,C 180,E1 -27506.101,E2 -27506.101} C_VEL
LIN {X 0,Y 115.754,Z 482.974,A -85,B 0,C 180,E1 -27510.94,E2 -27510.94} C_VEL
LIN {X 0,Y 115.015,Z 477.209,A -85,B 0,C 180,E1 -27515.681,E2 -27515.681} C_VEL
LIN {X 0,Y 114.615,Z 474.078,A -85,B 0,C 180,E1 -27518.413,E2 -27518.413} C_VEL
LIN {X 0,Y 114.026,Z 470.506,A -85,B 0,C 180,E1 -27522.051,E2 -27522.051} C_VEL
LIN {X 0,Y 112.938,Z 465.164,A -85,B 0,C 180,E1 -27529.241,E2 -27529.241} C_VEL
LIN {X 0,Y 112.393,Z 460.977,A -85,B 0,C 180,E1 -27540,E2 -27540} C_VEL
LIN {X 0,Y 112.644,Z 463.121,A -85,B 0,C 180,E1 -27550.788,E2 -27550.788} C_VEL
LIN {X 0,Y 113.123,Z 464.63,A -85,B 0,C 180,E1 -27554.389,E2 -27554.389} C_VEL
LIN {X 0,Y 114.124,Z 467.8,A -85,B 0,C 180,E1 -27559.798,E2 -27559.798} C_VEL
LIN {X 0,Y 115.011,Z 470.526,A -85,B 0,C 180,E1 -27563.565,E2 -27563.565} C_VEL
LIN {X 0,Y 116.251,Z 475.301,A -85,B 0,C 180,E1 -27568.924,E2 -27568.924} C_VEL
LIN {X 0,Y 117.349,Z 481.419,A -85,B 0,C 180,E1 -27574.676,E2 -27574.676} C_VEL
LIN {X 0,Y 117.599,Z 483.834,A -85,B 0,C 180,E1 -27576.7,E2 -27576.7} C_VEL
LIN {X 0,Y 117.187,Z 488.415,A -85,B 0,C 180,E1 -27580.004,E2 -27580.004} C_VEL
LIN {X 0,Y 116.735,Z 490.624,A -85,B 0,C 180,E1 -27581.472,E2 -27581.472} C_VEL
LIN {X 0,Y 115.904,Z 492.269,A -85,B 0,C 180,E1 -27582.34,E2 -27582.34} C_VEL
LIN {X 0,Y 110.17,Z 499.888,A -85,B 0,C 180,E1 -27585.901,E2 -27585.901} C_VEL
LIN {X 0,Y 106.806,Z 503.431,A -85,B 0,C 180,E1 -27587.685,E2 -27587.685} C_VEL
LIN {X 0,Y 99.95,Z 508.794,A -85,B 0,C 180,E1 -27590.342,E2 -27590.342} C_VEL
LIN {X 0,Y 93.096,Z 513.52,A -85,B 0,C 180,E1 -27593.55,E2 -27593.55} C_VEL
LIN {X 0,Y 89.868,Z 515.997,A -85,B 0,C 180,E1 -27596.21,E2 -27596.21} C_VEL
LIN {X 0,Y 84.958,Z 520.26,A -85,B 0,C 180,E1 -27602.937,E2 -27602.937} C_VEL
LIN {X 0,Y 81.507,Z 523.139,A -85,B 0,C 180,E1 -27609.824,E2 -27609.824} C_VEL
LIN {X 0,Y 78.706,Z 525.405,A -85,B 0,C 180,E1 -27619.187,E2 -27619.187} C_VEL
LIN {X 0,Y 77.84,Z 526.083,A -85,B 0,C 180,E1 -27624.82,E2 -27624.82} C_VEL
LIN {X 0,Y 77.612,Z 526.305,A -85,B 0,C 180,E1 -27630.001,E2 -27630.001} C_VEL
LIN {X 0,Y 77.832,Z 526.109,A -85,B 0,C 180,E1 -27635.181,E2 -27635.181} C_VEL
LIN {X 0,Y 78.576,Z 525.526,A -85,B 0,C 180,E1 -27640.305,E2 -27640.305} C_VEL
LIN {X 0,Y 81.44,Z 523.224,A -85,B 0,C 180,E1 -27650.194,E2 -27650.194} C_VEL
LIN {X 0,Y 84.915,Z 520.375,A -85,B 0,C 180,E1 -27657.079,E2 -27657.079} C_VEL
LIN {X 0,Y 89.448,Z 516.503,A -85,B 0,C 180,E1 -27663.367,E2 -27663.367} C_VEL
LIN {X 0,Y 94.893,Z 511.501,A -85,B 0,C 180,E1 -27669.017,E2 -27669.017} C_VEL
LIN {X 0,Y 101.025,Z 505.197,A -85,B 0,C 180,E1 -27674.081,E2 -27674.081} C_VEL
LIN {X 0,Y 107.927,Z 497.296,A -85,B 0,C 180,E1 -27678.493,E2 -27678.493} C_VEL
LIN {X 0,Y 110.32,Z 494.269,A -85,B 0,C 180,E1 -27679.86,E2 -27679.86} C_VEL
LIN {X 0,Y 111.29,Z 492.511,A -85,B 0,C 180,E1 -27680.838,E2 -27680.838} C_VEL
LIN {X 0,Y 111.989,Z 489.159,A -85,B 0,C 180,E1 -27683.405,E2 -27683.405} C_VEL
LIN {X 0,Y 111.984,Z 485.31,A -85,B 0,C 180,E1 -27686.912,E2 -27686.912} C_VEL
LIN {X 0,Y 111.441,Z 480.438,A -85,B 0,C 180,E1 -27691.996,E2 -27691.996} C_VEL
LIN {X 0,Y 110.982,Z 477.656,A -85,B 0,C 180,E1 -27695.247,E2 -27695.247} C_VEL
LIN {X 0,Y 110.063,Z 473.371,A -85,B 0,C 180,E1 -27701.381,E2 -27701.381} C_VEL
LIN {X 0,Y 109.592,Z 471.344,A -85,B 0,C 180,E1 -27705.136,E2 -27705.136} C_VEL
LIN {X 0,Y 109.218,Z 469.757,A -85,B 0,C 180,E1 -27708.869,E2 -27708.869} C_VEL
LIN {X 0,Y 108.899,Z 468.116,A -85,B 0,C 180,E1 -27716.3,E2 -27716.3} C_VEL
LIN {X 0,Y 109.131,Z 467.714,A -85,B 0,C 180,E1 -27720,E2 -27720} C_VEL
LIN {X 0,Y 109.072,Z 470.252,A -85,B 0,C 180,E1 -27727.404,E2 -27727.404} C_VEL
LIN {X 0,Y 109.416,Z 471.969,A -85,B 0,C 180,E1 -27731.11,E2 -27731.11} C_VEL
LIN {X 0,Y 109.92,Z 476.668,A -85,B 0,C 180,E1 -27737.463,E2 -27737.463} C_VEL
LIN {X 0,Y 110.302,Z 480.38,A -85,B 0,C 180,E1 -27741.492,E2 -27741.492} C_VEL
LIN {X 0,Y 110.662,Z 486.656,A -85,B 0,C 180,E1 -27747.235,E2 -27747.235} C_VEL
LIN {X 0,Y 110.651,Z 491.829,A -85,B 0,C 180,E1 -27751.426,E2 -27751.426} C_VEL
LIN {X 0,Y 110.493,Z 493.14,A -85,B 0,C 180,E1 -27752.374,E2 -27752.374} C_VEL
LIN {X 0,Y 107.575,Z 499.921,A -85,B 0,C 180,E1 -27756.014,E2 -27756.014} C_VEL
LIN {X 0,Y 102.805,Z 508.578,A -85,B 0,C 180,E1 -27761.236,E2 -27761.236} C_VEL
LIN {X 0,Y 99.595,Z 512.533,A -85,B 0,C 180,E1 -27763.671,E2 -27763.671} C_VEL
LIN {X 0,Y 94.246,Z 518.219,A -85,B 0,C 180,E1 -27767.844,E2 -27767.844} C_VEL
LIN {X 0,Y 88.725,Z 523.796,A -85,B 0,C 180,E1 -27773.552,E2 -27773.552} C_VEL
LIN {X 0,Y 84.01,Z 528.174,A -85,B 0,C 180,E1 -27779.871,E2 -27779.871} C_VEL
LIN {X 0,Y 81.432,Z 530.498,A -85,B 0,C 180,E1 -27784.435,E2 -27784.435} C_VEL
LIN {X 0,Y 79.522,Z 532.395,A -85,B 0,C 180,E1 -27789.297,E2 -27789.297} C_VEL
LIN {X 0,Y 77.353,Z 534.859,A -85,B 0,C 180,E1 -27799.53,E2 -27799.53} C_VEL
LIN {X 0,Y 77.068,Z 535.499,A -85,B 0,C 180,E1 -27804.767,E2 -27804.767} C_VEL
LIN {X 0,Y 77.278,Z 535.738,A -85,B 0,C 180,E1 -27809.999,E2 -27809.999} C_VEL
LIN {X 0,Y 77.067,Z 535.483,A -85,B 0,C 180,E1 -27815.232,E2 -27815.232} C_VEL
LIN {X 0,Y 77.346,Z 534.833,A -85,B 0,C 180,E1 -27820.47,E2 -27820.47} C_VEL
LIN {X 0,Y 79.518,Z 532.343,A -85,B 0,C 180,E1 -27830.703,E2 -27830.703} C_VEL
LIN {X 0,Y 82.669,Z 529.337,A -85,B 0,C 180,E1 -27837.877,E2 -27837.877} C_VEL
LIN {X 0,Y 87.007,Z 525.297,A -85,B 0,C 180,E1 -27844.431,E2 -27844.431} C_VEL
LIN {X 0,Y 92.352,Z 520.012,A -85,B 0,C 180,E1 -27850.447,E2 -27850.447} C_VEL
LIN {X 0,Y 98.47,Z 513.603,A -85,B 0,C 180,E1 -27855.538,E2 -27855.538} C_VEL
LIN {X 0,Y 101.811,Z 509.77,A -85,B 0,C 180,E1 -27857.908,E2 -27857.908} C_VEL
LIN {X 0,Y 105.357,Z 503.891,A -85,B 0,C 180,E1 -27861.61,E2 -27861.61} C_VEL
LIN {X 0,Y 109.581,Z 495.104,A -85,B 0,C 180,E1 -27866.487,E2 -27866.487} C_VEL
LIN {X 0,Y 110.486,Z 492.709,A -85,B 0,C 180,E1 -27867.747,E2 -27867.747} C_VEL
LIN {X 0,Y 110.557,Z 486.318,A -85,B 0,C 180,E1 -27872.869,E2 -27872.869} C_VEL
LIN {X 0,Y 110.127,Z 480.255,A -85,B 0,C 180,E1 -27878.472,E2 -27878.472} C_VEL
LIN {X 0,Y 109.821,Z 476.257,A -85,B 0,C 180,E1 -27882.682,E2 -27882.682} C_VEL
LIN {X 0,Y 109.288,Z 471.711,A -85,B 0,C 180,E1 -27888.877,E2 -27888.877} C_VEL
LIN {X 0,Y 108.948,Z 469.973,A -85,B 0,C 180,E1 -27892.587,E2 -27892.587} C_VEL
LIN {X 0,Y 109.032,Z 467.34,A -85,B 0,C 180,E1 -27900,E2 -27900} C_VEL
LIN {X 0,Y 108.771,Z 468.667,A -85,B 0,C 180,E1 -27907.874,E2 -27907.874} C_VEL
LIN {X 0,Y 109.064,Z 469.485,A -85,B 0,C 180,E1 -27911.147,E2 -27911.147} C_VEL
LIN {X 0,Y 109.474,Z 471.54,A -85,B 0,C 180,E1 -27915.641,E2 -27915.641} C_VEL
LIN {X 0,Y 110.158,Z 474.35,A -85,B 0,C 180,E1 -27920.542,E2 -27920.542} C_VEL
LIN {X 0,Y 110.757,Z 477.253,A -85,B 0,C 180,E1 -27924.528,E2 -27924.528} C_VEL
LIN {X 0,Y 111.351,Z 480.019,A -85,B 0,C 180,E1 -27927.918,E2 -27927.918} C_VEL
LIN {X 0,Y 111.901,Z 484.899,A -85,B 0,C 180,E1 -27933.004,E2 -27933.004} C_VEL
LIN {X 0,Y 112.05,Z 487.411,A -85,B 0,C 180,E1 -27935.375,E2 -27935.375} C_VEL
LIN {X 0,Y 111.214,Z 492.263,A -85,B 0,C 180,E1 -27939.193,E2 -27939.193} C_VEL
LIN {X 0,Y 110.355,Z 493.928,A -85,B 0,C 180,E1 -27940.162,E2 -27940.162} C_VEL
LIN {X 0,Y 103.33,Z 502.493,A -85,B 0,C 180,E1 -27944.426,E2 -27944.426} C_VEL
LIN {X 0,Y 96.909,Z 509.317,A -85,B 0,C 180,E1 -27949.255,E2 -27949.255} C_VEL
LIN {X 0,Y 91.224,Z 514.774,A -85,B 0,C 180,E1 -27954.704,E2 -27954.704} C_VEL
LIN {X 0,Y 89.868,Z 515.997,A -85,B 0,C 180,E1 -27956.21,E2 -27956.21} C_VEL
LIN {X 0,Y 86.796,Z 518.311,A -85,B 0,C 180,E1 -27959.123,E2 -27959.123} C_VEL
LIN {X 0,Y 80.607,Z 521.592,A -85,B 0,C 180,E1 -27963.934,E2 -27963.934} C_VEL
LIN {X 0,Y 75.907,Z 523.626,A -85,B 0,C 180,E1 -27968.388,E2 -27968.388} C_VEL
LIN {X 0,Y 73.351,Z 524.764,A -85,B 0,C 180,E1 -27972.394,E2 -27972.394} C_VEL
LIN {X 0,Y 72.812,Z 525.058,A -85,B 0,C 180,E1 -27973.865,E2 -27973.865} C_VEL
LIN {X 0,Y 70.808,Z 526.514,A -85,B 0,C 180,E1 -27984.304,E2 -27984.304} C_VEL
LIN {X 0,Y 70.527,Z 526.736,A -85,B 0,C 180,E1 -27990.001,E2 -27990.001} C_VEL
LIN {X 0,Y 71.319,Z 526.173,A -85,B 0,C 180,E1 -27999.789,E2 -27999.789} C_VEL
LIN {X 0,Y 72.957,Z 524.999,A -85,B 0,C 180,E1 -28006.798,E2 -28006.798} C_VEL
LIN {X 0,Y 74.832,Z 523.654,A -85,B 0,C 180,E1 -28012.066,E2 -28012.066} C_VEL
LIN {X 0,Y 78.66,Z 520.807,A -85,B 0,C 180,E1 -28019.434,E2 -28019.434} C_VEL
LIN {X 0,Y 83.631,Z 516.932,A -85,B 0,C 180,E1 -28026.034,E2 -28026.034} C_VEL
LIN {X 0,Y 89.504,Z 511.93,A -85,B 0,C 180,E1 -28031.87,E2 -28031.87} C_VEL
LIN {X 0,Y 96.075,Z 505.625,A -85,B 0,C 180,E1 -28037.014,E2 -28037.014} C_VEL
LIN {X 0,Y 103.377,Z 497.724,A -85,B 0,C 180,E1 -28041.428,E2 -28041.428} C_VEL
LIN {X 0,Y 105.712,Z 494.716,A -85,B 0,C 180,E1 -28042.921,E2 -28042.921} C_VEL
LIN {X 0,Y 106.481,Z 491.376,A -85,B 0,C 180,E1 -28045.873,E2 -28045.873} C_VEL
LIN {X 0,Y 106.479,Z 487.05,A -85,B 0,C 180,E1 -28050.566,E2 -28050.566} C_VEL
LIN {X 0,Y 106.314,Z 483.752,A -85,B 0,C 180,E1 -28054.552,E2 -28054.552} C_VEL
LIN {X 0,Y 105.767,Z 479.711,A -85,B 0,C 180,E1 -28060.595,E2 -28060.595} C_VEL
LIN {X 0,Y 105.524,Z 477.527,A -85,B 0,C 180,E1 -28064.549,E2 -28064.549} C_VEL
LIN {X 0,Y 105.269,Z 475.934,A -85,B 0,C 180,E1 -28068.446,E2 -28068.446} C_VEL
LIN {X 0,Y 105.091,Z 474.871,A -85,B 0,C 180,E1 -28072.313,E2 -28072.313} C_VEL
LIN {X 0,Y 105.128,Z 474.198,A -85,B 0,C 180,E1 -28076.167,E2 -28076.167} C_VEL
LIN {X 0,Y 105.406,Z 473.861,A -85,B 0,C 180,E1 -28080,E2 -28080} C_VEL
LIN {X 0,Y 105.173,Z 476.444,A -85,B 0,C 180,E1 -28087.68,E2 -28087.68} C_VEL
LIN {X 0,Y 105.307,Z 478.418,A -85,B 0,C 180,E1 -28091.549,E2 -28091.549} C_VEL
LIN {X 0,Y 105.437,Z 481.04,A -85,B 0,C 180,E1 -28095.463,E2 -28095.463} C_VEL
LIN {X 0,Y 105.52,Z 484.3,A -85,B 0,C 180,E1 -28099.452,E2 -28099.452} C_VEL
LIN {X 0,Y 105.409,Z 490.462,A -85,B 0,C 180,E1 -28105.682,E2 -28105.682} C_VEL
LIN {X 0,Y 105.106,Z 494.86,A -85,B 0,C 180,E1 -28109.626,E2 -28109.626} C_VEL
LIN {X 0,Y 104.557,Z 496.709,A -85,B 0,C 180,E1 -28110.964,E2 -28110.964} C_VEL
LIN {X 0,Y 100.825,Z 503.644,A -85,B 0,C 180,E1 -28115.011,E2 -28115.011} C_VEL
LIN {X 0,Y 97.068,Z 509.519,A -85,B 0,C 180,E1 -28118.891,E2 -28118.891} C_VEL
LIN {X 0,Y 93.623,Z 513.344,A -85,B 0,C 180,E1 -28121.351,E2 -28121.351} C_VEL
LIN {X 0,Y 86.531,Z 520.169,A -85,B 0,C 180,E1 -28126.968,E2 -28126.968} C_VEL
LIN {X 0,Y 81.228,Z 524.965,A -85,B 0,C 180,E1 -28132.723,E2 -28132.723} C_VEL
LIN {X 0,Y 76.443,Z 528.978,A -85,B 0,C 180,E1 -28139.624,E2 -28139.624} C_VEL
LIN {X 0,Y 72.884,Z 531.96,A -85,B 0,C 180,E1 -28147.312,E2 -28147.312} C_VEL
LIN {X 0,Y 70.353,Z 534.425,A -85,B 0,C 180,E1 -28158.475,E2 -28158.475} C_VEL
LIN {X 0,Y 69.989,Z 535.066,A -85,B 0,C 180,E1 -28164.236,E2 -28164.236} C_VEL
LIN {X 0,Y 70.193,Z 535.307,A -85,B 0,C 180,E1 -28169.999,E2 -28169.999} C_VEL
LIN {X 0,Y 69.988,Z 535.05,A -85,B 0,C 180,E1 -28175.763,E2 -28175.763} C_VEL
LIN {X 0,Y 70.346,Z 534.398,A -85,B 0,C 180,E1 -28181.525,E2 -28181.525} C_VEL
LIN {X 0,Y 72.881,Z 531.907,A -85,B 0,C 180,E1 -28192.688,E2 -28192.688} C_VEL
LIN {X 0,Y 76.442,Z 528.903,A -85,B 0,C 180,E1 -28200.375,E2 -28200.375} C_VEL
LIN {X 0,Y 81.226,Z 524.861,A -85,B 0,C 180,E1 -28207.277,E2 -28207.277} C_VEL
LIN {X 0,Y 87.796,Z 518.867,A -85,B 0,C 180,E1 -28214.14,E2 -28214.14} C_VEL
LIN {X 0,Y 94.794,Z 511.922,A -85,B 0,C 180,E1 -28219.458,E2 -28219.458} C_VEL
LIN {X 0,Y 97.025,Z 509.318,A -85,B 0,C 180,E1 -28221.139,E2 -28221.139} C_VEL
LIN {X 0,Y 101.717,Z 501.775,A -85,B 0,C 180,E1 -28226.009,E2 -28226.009} C_VEL
LIN {X 0,Y 104.479,Z 496.487,A -85,B 0,C 180,E1 -28229.057,E2 -28229.057} C_VEL
LIN {X 0,Y 105.009,Z 494.568,A -85,B 0,C 180,E1 -28230.465,E2 -28230.465} C_VEL
LIN {X 0,Y 105.301,Z 489.195,A -85,B 0,C 180,E1 -28235.346,E2 -28235.346} C_VEL
LIN {X 0,Y 105.372,Z 484.137,A -85,B 0,C 180,E1 -28240.52,E2 -28240.52} C_VEL
LIN {X 0,Y 105.312,Z 480.834,A -85,B 0,C 180,E1 -28244.518,E2 -28244.518} C_VEL
LIN {X 0,Y 105.19,Z 478.169,A -85,B 0,C 180,E1 -28248.438,E2 -28248.438} C_VEL
LIN {X 0,Y 105.062,Z 476.176,A -85,B 0,C 180,E1 -28252.312,E2 -28252.312} C_VEL
LIN {X 0,Y 105.318,Z 473.52,A -85,B 0,C 180,E1 -28260,E2 -28260} C_VEL
LIN {X 0,Y 105.018,Z 473.902,A -85,B 0,C 180,E1 -28263.837,E2 -28263.837} C_VEL
LIN {X 0,Y 104.941,Z 474.667,A -85,B 0,C 180,E1 -28267.861,E2 -28267.861} C_VEL
LIN {X 0,Y 105.115,Z 475.687,A -85,B 0,C 180,E1 -28271.571,E2 -28271.571} C_VEL
LIN {X 0,Y 105.484,Z 478.31,A -85,B 0,C 180,E1 -28277.447,E2 -28277.447} C_VEL
LIN {X 0,Y 105.884,Z 480.818,A -85,B 0,C 180,E1 -28281.683,E2 -28281.683} C_VEL
LIN {X 0,Y 106.207,Z 483.475,A -85,B 0,C 180,E1 -28285.476,E2 -28285.476} C_VEL
LIN {X 0,Y 106.466,Z 488.933,A -85,B 0,C 180,E1 -28291.877,E2 -28291.877} C_VEL
LIN {X 0,Y 106.448,Z 491.054,A -85,B 0,C 180,E1 -28294.139,E2 -28294.139} C_VEL
LIN {X 0,Y 105.657,Z 494.389,A -85,B 0,C 180,E1 -28297.041,E2 -28297.041} C_VEL
LIN {X 0,Y 104.979,Z 495.564,A -85,B 0,C 180,E1 -28297.737,E2 -28297.737} C_VEL
LIN {X 0,Y 97.301,Z 504.149,A -85,B 0,C 180,E1 -28302.239,E2 -28302.239} C_VEL
LIN {X 0,Y 91.651,Z 509.751,A -85,B 0,C 180,E1 -28306.359,E2 -28306.359} C_VEL
LIN {X 0,Y 85.534,Z 515.207,A -85,B 0,C 180,E1 -28311.958,E2 -28311.958} C_VEL
LIN {X 0,Y 80.242,Z 519.484,A -85,B 0,C 180,E1 -28318.298,E2 -28318.298} C_VEL
LIN {X 0,Y 77.305,Z 521.742,A -85,B 0,C 180,E1 -28322.964,E2 -28322.964} C_VEL
LIN {X 0,Y 74.883,Z 523.572,A -85,B 0,C 180,E1 -28327.951,E2 -28327.951} C_VEL
LIN {X 0,Y 72.812,Z 525.058,A -85,B 0,C 180,E1 -28333.865,E2 -28333.865} C_VEL
LIN {X 0,Y 71.019,Z 525.937,A -85,B 0,C 180,E1 -28338.314,E2 -28338.314} C_VEL
LIN {X 0,Y 67.083,Z 526.849,A -85,B 0,C 180,E1 -28345.851,E2 -28345.851} C_VEL
LIN {X 0,Y 64.557,Z 527.123,A -85,B 0,C 180,E1 -28352.453,E2 -28352.453} C_VEL
LIN {X 0,Y 63.959,Z 526.904,A -85,B 0,C 180,E1 -28357.729,E2 -28357.729} C_VEL
LIN {X 0,Y 64.129,Z 526.733,A -85,B 0,C 180,E1 -28359.49,E2 -28359.49} C_VEL
LIN {X 0,Y 66.209,Z 525.43,A -85,B 0,C 180,E1 -28368.57,E2 -28368.57} C_VEL
LIN {X 0,Y 68.331,Z 524.084,A -85,B 0,C 180,E1 -28374.294,E2 -28374.294} C_VEL
LIN {X 0,Y 72.568,Z 521.238,A -85,B 0,C 180,E1 -28382.186,E2 -28382.186} C_VEL
LIN {X 0,Y 78.009,Z 517.363,A -85,B 0,C 180,E1 -28389.098,E2 -28389.098} C_VEL
LIN {X 0,Y 84.344,Z 512.361,A -85,B 0,C 180,E1 -28395.095,E2 -28395.095} C_VEL
LIN {X 0,Y 91.405,Z 506.053,A -85,B 0,C 180,E1 -28400.255,E2 -28400.255} C_VEL
LIN {X 0,Y 99.627,Z 497.585,A -85,B 0,C 180,E1 -28404.891,E2 -28404.891} C_VEL
LIN {X 0,Y 100.511,Z 496.109,A -85,B 0,C 180,E1 -28405.987,E2 -28405.987} C_VEL
LIN {X 0,Y 100.945,Z 493.518,A -85,B 0,C 180,E1 -28408.842,E2 -28408.842} C_VEL
LIN {X 0,Y 101.217,Z 488.463,A -85,B 0,C 180,E1 -28415.379,E2 -28415.379} C_VEL
LIN {X 0,Y 101.061,Z 484.618,A -85,B 0,C 180,E1 -28421.763,E2 -28421.763} C_VEL
LIN {X 0,Y 100.976,Z 481.886,A -85,B 0,C 180,E1 -28427.948,E2 -28427.948} C_VEL
LIN {X 0,Y 100.917,Z 480.75,A -85,B 0,C 180,E1 -28431.993,E2 -28431.993} C_VEL
LIN {X 0,Y 101.012,Z 480.059,A -85,B 0,C 180,E1 -28436.01,E2 -28436.01} C_VEL
LIN {X 0,Y 101.303,Z 479.768,A -85,B 0,C 180,E1 -28440,E2 -28440} C_VEL
LIN {X 0,Y 100.981,Z 480.949,A -85,B 0,C 180,E1 -28443.991,E2 -28443.991} C_VEL
LIN {X 0,Y 100.877,Z 483.457,A -85,B 0,C 180,E1 -28450.03,E2 -28450.03} C_VEL
